LIN {X 0,Y 252.868,Z 364.586,A -85,B 0,C 180,E1 -18829.096,E2 -18829.096} C_VEL
LIN {X 0,Y 254.685,Z 356.199,A -85,B 0,C 180,E1 -18831.021,E2 -18831.021} C_VEL
LIN {X 0,Y 256.996,Z 345.688,A -85,B 0,C 180,E1 -18832.934,E2 -18832.934} C_VEL
LIN {X 0,Y 259.32,Z 333.859,A -85,B 0,C 180,E1 -18834.624,E2 -18834.624} C_VEL
LIN {X 0,Y 261.309,Z 321.945,A -85,B 0,C 180,E1 -18835.914,E2 -18835.914} C_VEL
LIN {X 0,Y 263.017,Z 309.547,A -85,B 0,C 180,E1 -18836.908,E2 -18836.908} C_VEL
LIN {X 0,Y 264.329,Z 296.774,A -85,B 0,C 180,E1 -18837.62,E2 -18837.62} C_VEL
LIN {X 0,Y 265.037,Z 283.246,A -85,B 0,C 180,E1 -18838.077,E2 -18838.077} C_VEL
LIN {X 0,Y 266.594,Z 234.638,A -85,B 0,C 180,E1 -18839.358,E2 -18839.358} C_VEL
LIN {X 0,Y 262.492,Z 206.676,A -85,B 0,C 180,E1 -18840.723,E2 -18840.723} C_VEL
LIN {X 0,Y 261.328,Z 202.665,A -85,B 0,C 180,E1 -18840.998,E2 -18840.998} C_VEL
LIN {X 0,Y 254.314,Z 186.379,A -85,B 0,C 180,E1 -18842.473,E2 -18842.473} C_VEL
LIN {X 0,Y 252.675,Z 182.594,A -85,B 0,C 180,E1 -18842.867,E2 -18842.867} C_VEL
LIN {X 0,Y 250.564,Z 173.371,A -85,B 0,C 180,E1 -18846.585,E2 -18846.585} C_VEL
LIN {X 0,Y 249.019,Z 167.461,A -85,B 0,C 180,E1 -18849.158,E2 -18849.158} C_VEL
LIN {X 0,Y 248.966,Z 167.471,A -85,B 0,C 180,E1 -18852.781,E2 -18852.781} C_VEL
LIN {X 0,Y 248.974,Z 167.471,A -85,B 0,C 180,E1 -18857.354,E2 -18857.354} C_VEL
LIN {X 0,Y 249.034,Z 167.462,A -85,B 0,C 180,E1 -18862.201,E2 -18862.201} C_VEL
LIN {X 0,Y 249.037,Z 167.461,A -85,B 0,C 180,E1 -18865.638,E2 -18865.638} C_VEL
LIN {X 0,Y 248.996,Z 167.466,A -85,B 0,C 180,E1 -18869.465,E2 -18869.465} C_VEL
LIN {X 0,Y 249.015,Z 167.464,A -85,B 0,C 180,E1 -18873.155,E2 -18873.155} C_VEL
LIN {X 0,Y 248.999,Z 167.459,A -85,B 0,C 180,E1 -18876.725,E2 -18876.725} C_VEL
LIN {X 0,Y 249.035,Z 167.464,A -85,B 0,C 180,E1 -18880.205,E2 -18880.205} C_VEL
LIN {X 0,Y 249.151,Z 167.437,A -85,B 0,C 180,E1 -18883.616,E2 -18883.616} C_VEL
LIN {X 0,Y 249.21,Z 167.436,A -85,B 0,C 180,E1 -18888.615,E2 -18888.615} C_VEL
LIN {X 0,Y 249.394,Z 167.413,A -85,B 0,C 180,E1 -18891.9,E2 -18891.9} C_VEL
LIN {X 0,Y 249.245,Z 167.435,A -85,B 0,C 180,E1 -18895.148,E2 -18895.148} C_VEL
LIN {X 0,Y 249.646,Z 167.378,A -85,B 0,C 180,E1 -18898.387,E2 -18898.387} C_VEL
LIN {X 0,Y 249.648,Z 167.388,A -85,B 0,C 180,E1 -18901.613,E2 -18901.613} C_VEL
LIN {X 0,Y 249.415,Z 167.411,A -85,B 0,C 180,E1 -18906.557,E2 -18906.557} C_VEL
LIN {X 0,Y 249.325,Z 167.427,A -85,B 0,C 180,E1 -18909.737,E2 -18909.737} C_VEL
LIN {X 0,Y 249.139,Z 167.448,A -85,B 0,C 180,E1 -18914.708,E2 -18914.708} C_VEL
LIN {X 0,Y 249.073,Z 167.452,A -85,B 0,C 180,E1 -18918.082,E2 -18918.082} C_VEL
LIN {X 0,Y 249.039,Z 167.461,A -85,B 0,C 180,E1 -18921.523,E2 -18921.523} C_VEL
LIN {X 0,Y 249.056,Z 167.452,A -85,B 0,C 180,E1 -18925.449,E2 -18925.449} C_VEL
LIN {X 0,Y 249.03,Z 167.466,A -85,B 0,C 180,E1 -18928.974,E2 -18928.974} C_VEL
LIN {X 0,Y 249.022,Z 167.458,A -85,B 0,C 180,E1 -18932.427,E2 -18932.427} C_VEL
LIN {X 0,Y 249.021,Z 167.465,A -85,B 0,C 180,E1 -18936.347,E2 -18936.347} C_VEL
LIN {X 0,Y 248.974,Z 167.47,A -85,B 0,C 180,E1 -18940.485,E2 -18940.485} C_VEL
LIN {X 0,Y 248.978,Z 167.466,A -85,B 0,C 180,E1 -18944.885,E2 -18944.885} C_VEL
LIN {X 0,Y 249.003,Z 167.467,A -85,B 0,C 180,E1 -18947.362,E2 -18947.362} C_VEL
LIN {X 0,Y 249.039,Z 167.461,A -85,B 0,C 180,E1 -18952.202,E2 -18952.202} C_VEL
LIN {X 0,Y 249.028,Z 167.546,A -85,B 0,C 180,E1 -18956.659,E2 -18956.659} C_VEL
LIN {X 0,Y 250.144,Z 170.47,A -85,B 0,C 180,E1 -18956.949,E2 -18956.949} C_VEL
LIN {X 0,Y 251.527,Z 172.737,A -85,B 0,C 180,E1 -18957.231,E2 -18957.231} C_VEL
LIN {X 0,Y 257.093,Z 183.362,A -85,B 0,C 180,E1 -18958.378,E2 -18958.378} C_VEL
LIN {X 0,Y 264.699,Z 200.479,A -85,B 0,C 180,E1 -18959.926,E2 -18959.926} C_VEL
LIN {X 0,Y 267.489,Z 207.786,A -85,B 0,C 180,E1 -18960.497,E2 -18960.497} C_VEL
LIN {X 0,Y 265.356,Z 271.347,A -85,B 0,C 180,E1 -18962.177,E2 -18962.177} C_VEL
LIN {X 0,Y 264.517,Z 284.387,A -85,B 0,C 180,E1 -18962.724,E2 -18962.724} C_VEL
LIN {X 0,Y 263.3,Z 296.87,A -85,B 0,C 180,E1 -18963.551,E2 -18963.551} C_VEL
LIN {X 0,Y 261.894,Z 308.06,A -85,B 0,C 180,E1 -18964.574,E2 -18964.574} C_VEL
LIN {X 0,Y 260.057,Z 319.137,A -85,B 0,C 180,E1 -18965.875,E2 -18965.875} C_VEL
LIN {X 0,Y 258.172,Z 329.268,A -85,B 0,C 180,E1 -18967.388,E2 -18967.388} C_VEL
LIN {X 0,Y 256.493,Z 338.564,A -85,B 0,C 180,E1 -18969.134,E2 -18969.134} C_VEL
LIN {X 0,Y 254.459,Z 347.043,A -85,B 0,C 180,E1 -18971.064,E2 -18971.064} C_VEL
LIN {X 0,Y 252.372,Z 355.282,A -85,B 0,C 180,E1 -18973.416,E2 -18973.416} C_VEL
LIN {X 0,Y 250.964,Z 360.914,A -85,B 0,C 180,E1 -18975.403,E2 -18975.403} C_VEL
LIN {X 0,Y 249.579,Z 366.401,A -85,B 0,C 180,E1 -18977.809,E2 -18977.809} C_VEL
LIN {X 0,Y 248.492,Z 370.708,A -85,B 0,C 180,E1 -18980.231,E2 -18980.231} C_VEL
LIN {X 0,Y 247.724,Z 374.525,A -85,B 0,C 180,E1 -18983.2,E2 -18983.2} C_VEL
LIN {X 0,Y 247.414,Z 376.22,A -85,B 0,C 180,E1 -18985.112,E2 -18985.112} C_VEL
LIN {X 0,Y 247.22,Z 377.209,A -85,B 0,C 180,E1 -18986.742,E2 -18986.742} C_VEL
LIN {X 0,Y 247.041,Z 378.047,A -85,B 0,C 180,E1 -18990.001,E2 -18990.001} C_VEL
LIN {X 0,Y 247.079,Z 377.854,A -85,B 0,C 180,E1 -18991.631,E2 -18991.631} C_VEL
LIN {X 0,Y 247.218,Z 377.268,A -85,B 0,C 180,E1 -18993.26,E2 -18993.26} C_VEL
LIN {X 0,Y 247.408,Z 376.303,A -85,B 0,C 180,E1 -18994.889,E2 -18994.889} C_VEL
LIN {X 0,Y 247.716,Z 374.678,A -85,B 0,C 180,E1 -18996.784,E2 -18996.784} C_VEL
LIN {X 0,Y 248.467,Z 370.899,A -85,B 0,C 180,E1 -18999.772,E2 -18999.772} C_VEL
LIN {X 0,Y 249.523,Z 366.652,A -85,B 0,C 180,E1 -19002.196,E2 -19002.196} C_VEL
LIN {X 0,Y 251.213,Z 360.217,A -85,B 0,C 180,E1 -19004.998,E2 -19004.998} C_VEL
LIN {X 0,Y 252.923,Z 353.147,A -85,B 0,C 180,E1 -19007.381,E2 -19007.381} C_VEL
LIN {X 0,Y 255.176,Z 344.328,A -85,B 0,C 180,E1 -19009.718,E2 -19009.718} C_VEL
LIN {X 0,Y 257.073,Z 335.367,A -85,B 0,C 180,E1 -19011.641,E2 -19011.641} C_VEL
LIN {X 0,Y 259.036,Z 325.258,A -85,B 0,C 180,E1 -19013.379,E2 -19013.379} C_VEL
LIN {X 0,Y 261.004,Z 314.1,A -85,B 0,C 180,E1 -19014.881,E2 -19014.881} C_VEL
LIN {X 0,Y 262.591,Z 303.55,A -85,B 0,C 180,E1 -19015.993,E2 -19015.993} C_VEL
LIN {X 0,Y 264.079,Z 290.832,A -85,B 0,C 180,E1 -19017.007,E2 -19017.007} C_VEL
LIN {X 0,Y 265.098,Z 278.105,A -85,B 0,C 180,E1 -19017.696,E2 -19017.696} C_VEL
LIN {X 0,Y 265.964,Z 260.051,A -85,B 0,C 180,E1 -19018.24,E2 -19018.24} C_VEL
LIN {X 0,Y 267.533,Z 207.816,A -85,B 0,C 180,E1 -19019.63,E2 -19019.63} C_VEL
LIN {X 0,Y 261.17,Z 192.177,A -85,B 0,C 180,E1 -19020.926,E2 -19020.926} C_VEL
LIN {X 0,Y 254.413,Z 178.027,A -85,B 0,C 180,E1 -19022.313,E2 -19022.313} C_VEL
LIN {X 0,Y 250.64,Z 171.151,A -85,B 0,C 180,E1 -19023.096,E2 -19023.096} C_VEL
LIN {X 0,Y 249.295,Z 168.69,A -85,B 0,C 180,E1 -19023.383,E2 -19023.383} C_VEL
LIN {X 0,Y 249.029,Z 167.477,A -85,B 0,C 180,E1 -19023.515,E2 -19023.515} C_VEL
LIN {X 0,Y 249.04,Z 167.465,A -85,B 0,C 180,E1 -19027.798,E2 -19027.798} C_VEL
LIN {X 0,Y 248.978,Z 167.471,A -85,B 0,C 180,E1 -19032.646,E2 -19032.646} C_VEL
LIN {X 0,Y 248.98,Z 167.471,A -85,B 0,C 180,E1 -19037.355,E2 -19037.355} C_VEL
LIN {X 0,Y 249.041,Z 167.461,A -85,B 0,C 180,E1 -19042.201,E2 -19042.201} C_VEL
LIN {X 0,Y 249.044,Z 167.456,A -85,B 0,C 180,E1 -19045.639,E2 -19045.639} C_VEL
LIN {X 0,Y 249.003,Z 167.462,A -85,B 0,C 180,E1 -19049.466,E2 -19049.466} C_VEL
LIN {X 0,Y 249.036,Z 167.465,A -85,B 0,C 180,E1 -19053.158,E2 -19053.158} C_VEL
LIN {X 0,Y 249.056,Z 167.45,A -85,B 0,C 180,E1 -19056.73,E2 -19056.73} C_VEL
LIN {X 0,Y 249.076,Z 167.457,A -85,B 0,C 180,E1 -19060.208,E2 -19060.208} C_VEL
LIN {X 0,Y 249.158,Z 167.441,A -85,B 0,C 180,E1 -19063.616,E2 -19063.616} C_VEL
LIN {X 0,Y 249.229,Z 167.441,A -85,B 0,C 180,E1 -19068.615,E2 -19068.615} C_VEL
LIN {X 0,Y 249.417,Z 167.405,A -85,B 0,C 180,E1 -19071.901,E2 -19071.901} C_VEL
LIN {X 0,Y 249.258,Z 167.431,A -85,B 0,C 180,E1 -19075.148,E2 -19075.148} C_VEL
LIN {X 0,Y 249.655,Z 167.384,A -85,B 0,C 180,E1 -19078.387,E2 -19078.387} C_VEL
LIN {X 0,Y 249.653,Z 167.37,A -85,B 0,C 180,E1 -19081.613,E2 -19081.613} C_VEL
LIN {X 0,Y 249.252,Z 167.435,A -85,B 0,C 180,E1 -19084.802,E2 -19084.802} C_VEL
LIN {X 0,Y 248.58,Z 167.529,A -85,B 0,C 180,E1 -19086.153,E2 -19086.153} C_VEL
LIN {X 0,Y 245.744,Z 167.883,A -85,B 0,C 180,E1 -19088.356,E2 -19088.356} C_VEL
LIN {X 0,Y 243.315,Z 168.178,A -85,B 0,C 180,E1 -19090.15,E2 -19090.15} C_VEL
LIN {X 0,Y 242.234,Z 168.307,A -85,B 0,C 180,E1 -19091.541,E2 -19091.541} C_VEL
LIN {X 0,Y 242.125,Z 168.319,A -85,B 0,C 180,E1 -19092.013,E2 -19092.013} C_VEL
LIN {X 0,Y 242.092,Z 168.312,A -85,B 0,C 180,E1 -19096.876,E2 -19096.876} C_VEL
LIN {X 0,Y 241.972,Z 168.336,A -85,B 0,C 180,E1 -19102.184,E2 -19102.184} C_VEL
LIN {X 0,Y 241.987,Z 168.342,A -85,B 0,C 180,E1 -19105.826,E2 -19105.826} C_VEL
LIN {X 0,Y 241.968,Z 168.337,A -85,B 0,C 180,E1 -19109.589,E2 -19109.589} C_VEL
LIN {X 0,Y 241.98,Z 168.335,A -85,B 0,C 180,E1 -19113.493,E2 -19113.493} C_VEL
LIN {X 0,Y 241.978,Z 168.336,A -85,B 0,C 180,E1 -19117.584,E2 -19117.584} C_VEL
LIN {X 0,Y 241.908,Z 168.347,A -85,B 0,C 180,E1 -19121.929,E2 -19121.929} C_VEL
LIN {X 0,Y 241.901,Z 168.351,A -85,B 0,C 180,E1 -19126.58,E2 -19126.58} C_VEL
LIN {X 0,Y 241.977,Z 168.45,A -85,B 0,C 180,E1 -19129.989,E2 -19129.989} C_VEL
LIN {X 0,Y 244.385,Z 177.67,A -85,B 0,C 180,E1 -19134.066,E2 -19134.066} C_VEL
LIN {X 0,Y 245.43,Z 182.458,A -85,B 0,C 180,E1 -19136.022,E2 -19136.022} C_VEL
LIN {X 0,Y 253.06,Z 199.303,A -85,B 0,C 180,E1 -19137.723,E2 -19137.723} C_VEL
LIN {X 0,Y 256.555,Z 208.314,A -85,B 0,C 180,E1 -19138.499,E2 -19138.499} C_VEL
LIN {X 0,Y 260.098,Z 232.626,A -85,B 0,C 180,E1 -19139.735,E2 -19139.735} C_VEL
LIN {X 0,Y 260.446,Z 237.003,A -85,B 0,C 180,E1 -19139.915,E2 -19139.915} C_VEL
LIN {X 0,Y 258.519,Z 291.741,A -85,B 0,C 180,E1 -19141.425,E2 -19141.425} C_VEL
LIN {X 0,Y 257.264,Z 305.637,A -85,B 0,C 180,E1 -19142.106,E2 -19142.106} C_VEL
LIN {X 0,Y 255.612,Z 318.073,A -85,B 0,C 180,E1 -19143.021,E2 -19143.021} C_VEL
LIN {X 0,Y 253.774,Z 329.173,A -85,B 0,C 180,E1 -19144.139,E2 -19144.139} C_VEL
LIN {X 0,Y 251.513,Z 340.745,A -85,B 0,C 180,E1 -19145.659,E2 -19145.659} C_VEL
LIN {X 0,Y 249.22,Z 351.171,A -85,B 0,C 180,E1 -19147.404,E2 -19147.404} C_VEL
LIN {X 0,Y 247.242,Z 359.7,A -85,B 0,C 180,E1 -19149.186,E2 -19149.186} C_VEL
LIN {X 0,Y 245.437,Z 367.793,A -85,B 0,C 180,E1 -19151.272,E2 -19151.272} C_VEL
LIN {X 0,Y 243.537,Z 375.272,A -85,B 0,C 180,E1 -19153.658,E2 -19153.658} C_VEL
LIN {X 0,Y 241.694,Z 382.371,A -85,B 0,C 180,E1 -19156.548,E2 -19156.548} C_VEL
LIN {X 0,Y 240.787,Z 387.105,A -85,B 0,C 180,E1 -19159.063,E2 -19159.063} C_VEL
LIN {X 0,Y 240.158,Z 390.724,A -85,B 0,C 180,E1 -19161.585,E2 -19161.585} C_VEL
LIN {X 0,Y 239.899,Z 392.592,A -85,B 0,C 180,E1 -19163.27,E2 -19163.27} C_VEL
LIN {X 0,Y 239.798,Z 394.153,A -85,B 0,C 180,E1 -19165.188,E2 -19165.188} C_VEL
LIN {X 0,Y 239.883,Z 395.614,A -85,B 0,C 180,E1 -19168.32,E2 -19168.32} C_VEL
LIN {X 0,Y 239.956,Z 395.83,A -85,B 0,C 180,E1 -19169.999,E2 -19169.999} C_VEL
LIN {X 0,Y 239.883,Z 395.604,A -85,B 0,C 180,E1 -19171.678,E2 -19171.678} C_VEL
LIN {X 0,Y 239.78,Z 394.165,A -85,B 0,C 180,E1 -19174.76,E2 -19174.76} C_VEL
LIN {X 0,Y 239.905,Z 392.559,A -85,B 0,C 180,E1 -19176.728,E2 -19176.728} C_VEL
LIN {X 0,Y 240.359,Z 389.6,A -85,B 0,C 180,E1 -19179.253,E2 -19179.253} C_VEL
LIN {X 0,Y 241.052,Z 385.599,A -85,B 0,C 180,E1 -19181.775,E2 -19181.775} C_VEL
LIN {X 0,Y 242.451,Z 379.459,A -85,B 0,C 180,E1 -19184.692,E2 -19184.692} C_VEL
LIN {X 0,Y 244.066,Z 372.759,A -85,B 0,C 180,E1 -19187.166,E2 -19187.166} C_VEL
LIN {X 0,Y 245.951,Z 365.05,A -85,B 0,C 180,E1 -19189.444,E2 -19189.444} C_VEL
LIN {X 0,Y 248.049,Z 355.936,A -85,B 0,C 180,E1 -19191.611,E2 -19191.611} C_VEL
LIN {X 0,Y 250.431,Z 345.424,A -85,B 0,C 180,E1 -19193.571,E2 -19193.571} C_VEL
LIN {X 0,Y 252.885,Z 333.595,A -85,B 0,C 180,E1 -19195.294,E2 -19195.294} C_VEL
LIN {X 0,Y 254.951,Z 321.68,A -85,B 0,C 180,E1 -19196.611,E2 -19196.611} C_VEL
LIN {X 0,Y 256.725,Z 309.281,A -85,B 0,C 180,E1 -19197.623,E2 -19197.623} C_VEL
LIN {X 0,Y 258.064,Z 296.503,A -85,B 0,C 180,E1 -19198.35,E2 -19198.35} C_VEL
LIN {X 0,Y 258.784,Z 282.965,A -85,B 0,C 180,E1 -19198.818,E2 -19198.818} C_VEL
LIN {X 0,Y 260.307,Z 234.676,A -85,B 0,C 180,E1 -19200.13,E2 -19200.13} C_VEL
LIN {X 0,Y 256.425,Z 208.257,A -85,B 0,C 180,E1 -19201.472,E2 -19201.472} C_VEL
LIN {X 0,Y 254.062,Z 201.684,A -85,B 0,C 180,E1 -19202.009,E2 -19202.009} C_VEL
LIN {X 0,Y 246.909,Z 185.778,A -85,B 0,C 180,E1 -19203.582,E2 -19203.582} C_VEL
LIN {X 0,Y 245.392,Z 182.189,A -85,B 0,C 180,E1 -19204.005,E2 -19204.005} C_VEL
LIN {X 0,Y 243.08,Z 172.44,A -85,B 0,C 180,E1 -19208.142,E2 -19208.142} C_VEL
LIN {X 0,Y 241.946,Z 168.341,A -85,B 0,C 180,E1 -19210.074,E2 -19210.074} C_VEL
LIN {X 0,Y 241.892,Z 168.354,A -85,B 0,C 180,E1 -19214.209,E2 -19214.209} C_VEL
LIN {X 0,Y 241.903,Z 168.353,A -85,B 0,C 180,E1 -19218.07,E2 -19218.07} C_VEL
LIN {X 0,Y 241.977,Z 168.34,A -85,B 0,C 180,E1 -19222.416,E2 -19222.416} C_VEL
LIN {X 0,Y 241.973,Z 168.337,A -85,B 0,C 180,E1 -19226.506,E2 -19226.506} C_VEL
LIN {X 0,Y 241.971,Z 168.337,A -85,B 0,C 180,E1 -19230.612,E2 -19230.612} C_VEL
LIN {X 0,Y 241.99,Z 168.339,A -85,B 0,C 180,E1 -19234.196,E2 -19234.196} C_VEL
LIN {X 0,Y 241.978,Z 168.335,A -85,B 0,C 180,E1 -19238.338,E2 -19238.338} C_VEL
LIN {X 0,Y 242.099,Z 168.314,A -85,B 0,C 180,E1 -19243.324,E2 -19243.324} C_VEL
LIN {X 0,Y 242.144,Z 168.318,A -85,B 0,C 180,E1 -19248.278,E2 -19248.278} C_VEL
LIN {X 0,Y 242.35,Z 168.289,A -85,B 0,C 180,E1 -19251.663,E2 -19251.663} C_VEL
LIN {X 0,Y 242.382,Z 168.291,A -85,B 0,C 180,E1 -19253.34,E2 -19253.34} C_VEL
LIN {X 0,Y 242.606,Z 168.254,A -85,B 0,C 180,E1 -19258.34,E2 -19258.34} C_VEL
LIN {X 0,Y 242.608,Z 168.266,A -85,B 0,C 180,E1 -19261.66,E2 -19261.66} C_VEL
LIN {X 0,Y 242.392,Z 168.286,A -85,B 0,C 180,E1 -19266.66,E2 -19266.66} C_VEL
LIN {X 0,Y 242.253,Z 168.306,A -85,B 0,C 180,E1 -19270.024,E2 -19270.024} C_VEL
LIN {X 0,Y 242.097,Z 168.326,A -85,B 0,C 180,E1 -19275.145,E2 -19275.145} C_VEL
LIN {X 0,Y 242.012,Z 168.331,A -85,B 0,C 180,E1 -19278.629,E2 -19278.629} C_VEL
LIN {X 0,Y 241.978,Z 168.342,A -85,B 0,C 180,E1 -19282.183,E2 -19282.183} C_VEL
LIN {X 0,Y 241.987,Z 168.33,A -85,B 0,C 180,E1 -19285.826,E2 -19285.826} C_VEL
LIN {X 0,Y 241.963,Z 168.344,A -85,B 0,C 180,E1 -19289.589,E2 -19289.589} C_VEL
LIN {X 0,Y 241.974,Z 168.344,A -85,B 0,C 180,E1 -19293.494,E2 -19293.494} C_VEL
LIN {X 0,Y 241.978,Z 168.341,A -85,B 0,C 180,E1 -19297.584,E2 -19297.584} C_VEL
LIN {X 0,Y 241.908,Z 168.35,A -85,B 0,C 180,E1 -19301.929,E2 -19301.929} C_VEL
LIN {X 0,Y 241.919,Z 168.35,A -85,B 0,C 180,E1 -19306.575,E2 -19306.575} C_VEL
LIN {X 0,Y 241.991,Z 168.337,A -85,B 0,C 180,E1 -19311.642,E2 -19311.642} C_VEL
LIN {X 0,Y 242.041,Z 168.531,A -85,B 0,C 180,E1 -19315.609,E2 -19315.609} C_VEL
LIN {X 0,Y 243.04,Z 171.272,A -85,B 0,C 180,E1 -19315.868,E2 -19315.868} C_VEL
LIN {X 0,Y 244.462,Z 173.486,A -85,B 0,C 180,E1 -19316.173,E2 -19316.173} C_VEL
LIN {X 0,Y 249.703,Z 182.957,A -85,B 0,C 180,E1 -19317.302,E2 -19317.302} C_VEL
LIN {X 0,Y 256.513,Z 197.662,A -85,B 0,C 180,E1 -19318.758,E2 -19318.758} C_VEL
LIN {X 0,Y 261.307,Z 209.496,A -85,B 0,C 180,E1 -19319.771,E2 -19319.771} C_VEL
LIN {X 0,Y 259.135,Z 271.055,A -85,B 0,C 180,E1 -19321.428,E2 -19321.428} C_VEL
LIN {X 0,Y 258.314,Z 283.988,A -85,B 0,C 180,E1 -19321.971,E2 -19321.971} C_VEL
LIN {X 0,Y 257.098,Z 295.986,A -85,B 0,C 180,E1 -19322.751,E2 -19322.751} C_VEL
LIN {X 0,Y 255.523,Z 308.324,A -85,B 0,C 180,E1 -19323.893,E2 -19323.893} C_VEL
LIN {X 0,Y 253.592,Z 319.401,A -85,B 0,C 180,E1 -19325.219,E2 -19325.219} C_VEL
LIN {X 0,Y 251.628,Z 329.532,A -85,B 0,C 180,E1 -19326.766,E2 -19326.766} C_VEL
LIN {X 0,Y 249.869,Z 338.826,A -85,B 0,C 180,E1 -19328.554,E2 -19328.554} C_VEL
LIN {X 0,Y 247.752,Z 347.304,A -85,B 0,C 180,E1 -19330.531,E2 -19330.531} C_VEL
LIN {X 0,Y 245.588,Z 355.543,A -85,B 0,C 180,E1 -19332.944,E2 -19332.944} C_VEL
LIN {X 0,Y 244.098,Z 361.175,A -85,B 0,C 180,E1 -19334.983,E2 -19334.983} C_VEL
LIN {X 0,Y 242.646,Z 366.662,A -85,B 0,C 180,E1 -19337.455,E2 -19337.455} C_VEL
LIN {X 0,Y 241.503,Z 370.968,A -85,B 0,C 180,E1 -19339.945,E2 -19339.945} C_VEL
LIN {X 0,Y 240.976,Z 373.243,A -85,B 0,C 180,E1 -19341.616,E2 -19341.616} C_VEL
LIN {X 0,Y 240.601,Z 375.091,A -85,B 0,C 180,E1 -19343.291,E2 -19343.291} C_VEL
LIN {X 0,Y 240.334,Z 376.48,A -85,B 0,C 180,E1 -19344.968,E2 -19344.968} C_VEL
LIN {X 0,Y 240.142,Z 377.468,A -85,B 0,C 180,E1 -19346.645,E2 -19346.645} C_VEL
LIN {X 0,Y 239.971,Z 378.305,A -85,B 0,C 180,E1 -19350.001,E2 -19350.001} C_VEL
LIN {X 0,Y 240.012,Z 378.112,A -85,B 0,C 180,E1 -19351.679,E2 -19351.679} C_VEL
LIN {X 0,Y 240.139,Z 377.527,A -85,B 0,C 180,E1 -19353.356,E2 -19353.356} C_VEL
LIN {X 0,Y 240.329,Z 376.562,A -85,B 0,C 180,E1 -19355.034,E2 -19355.034} C_VEL
LIN {X 0,Y 240.602,Z 375.209,A -85,B 0,C 180,E1 -19356.711,E2 -19356.711} C_VEL
LIN {X 0,Y 241.197,Z 372.35,A -85,B 0,C 180,E1 -19359.223,E2 -19359.223} C_VEL
LIN {X 0,Y 242.16,Z 368.467,A -85,B 0,C 180,E1 -19361.722,E2 -19361.722} C_VEL
LIN {X 0,Y 243.536,Z 363.454,A -85,B 0,C 180,E1 -19364.2,E2 -19364.2} C_VEL
LIN {X 0,Y 245.157,Z 357.141,A -85,B 0,C 180,E1 -19366.66,E2 -19366.66} C_VEL
LIN {X 0,Y 247.326,Z 349.232,A -85,B 0,C 180,E1 -19369.074,E2 -19369.074} C_VEL
LIN {X 0,Y 249.737,Z 339.396,A -85,B 0,C 180,E1 -19371.46,E2 -19371.46} C_VEL
LIN {X 0,Y 251.803,Z 329.072,A -85,B 0,C 180,E1 -19373.437,E2 -19373.437} C_VEL
LIN {X 0,Y 254.091,Z 317.414,A -85,B 0,C 180,E1 -19375.168,E2 -19375.168} C_VEL
LIN {X 0,Y 256.028,Z 305.781,A -85,B 0,C 180,E1 -19376.492,E2 -19376.492} C_VEL
LIN {X 0,Y 257.504,Z 293.679,A -85,B 0,C 180,E1 -19377.534,E2 -19377.534} C_VEL
LIN {X 0,Y 258.64,Z 281.366,A -85,B 0,C 180,E1 -19378.284,E2 -19378.284} C_VEL
LIN {X 0,Y 259.432,Z 269.158,A -85,B 0,C 180,E1 -19378.741,E2 -19378.741} C_VEL
LIN {X 0,Y 261.376,Z 209.619,A -85,B 0,C 180,E1 -19380.352,E2 -19380.352} C_VEL
LIN {X 0,Y 254.384,Z 192.715,A -85,B 0,C 180,E1 -19381.837,E2 -19381.837} C_VEL
LIN {X 0,Y 247.191,Z 178.132,A -85,B 0,C 180,E1 -19383.385,E2 -19383.385} C_VEL
LIN {X 0,Y 243.415,Z 171.757,A -85,B 0,C 180,E1 -19384.201,E2 -19384.201} C_VEL
LIN {X 0,Y 242.12,Z 168.986,A -85,B 0,C 180,E1 -19384.509,E2 -19384.509} C_VEL
LIN {X 0,Y 242.017,Z 168.336,A -85,B 0,C 180,E1 -19384.643,E2 -19384.643} C_VEL
LIN {X 0,Y 241.986,Z 168.342,A -85,B 0,C 180,E1 -19388.356,E2 -19388.356} C_VEL
LIN {X 0,Y 241.9,Z 168.354,A -85,B 0,C 180,E1 -19393.42,E2 -19393.42} C_VEL
LIN {X 0,Y 241.909,Z 168.35,A -85,B 0,C 180,E1 -19398.071,E2 -19398.071} C_VEL
LIN {X 0,Y 241.984,Z 168.341,A -85,B 0,C 180,E1 -19402.417,E2 -19402.417} C_VEL
LIN {X 0,Y 241.98,Z 168.338,A -85,B 0,C 180,E1 -19406.507,E2 -19406.507} C_VEL
LIN {X 0,Y 241.978,Z 168.332,A -85,B 0,C 180,E1 -19410.613,E2 -19410.613} C_VEL
LIN {X 0,Y 242.033,Z 168.336,A -85,B 0,C 180,E1 -19414.179,E2 -19414.179} C_VEL
LIN {X 0,Y 242.023,Z 168.324,A -85,B 0,C 180,E1 -19418.316,E2 -19418.316} C_VEL
LIN {X 0,Y 242.106,Z 168.319,A -85,B 0,C 180,E1 -19423.324,E2 -19423.324} C_VEL
LIN {X 0,Y 242.161,Z 168.32,A -85,B 0,C 180,E1 -19428.278,E2 -19428.278} C_VEL
LIN {X 0,Y 242.371,Z 168.284,A -85,B 0,C 180,E1 -19431.664,E2 -19431.664} C_VEL
LIN {X 0,Y 242.395,Z 168.273,A -85,B 0,C 180,E1 -19433.34,E2 -19433.34} C_VEL
LIN {X 0,Y 242.615,Z 168.261,A -85,B 0,C 180,E1 -19438.34,E2 -19438.34} C_VEL
LIN {X 0,Y 242.613,Z 168.246,A -85,B 0,C 180,E1 -19441.66,E2 -19441.66} C_VEL
LIN {X 0,Y 242.389,Z 168.288,A -85,B 0,C 180,E1 -19446.66,E2 -19446.66} C_VEL
LIN {X 0,Y 242.259,Z 168.293,A -85,B 0,C 180,E1 -19450.024,E2 -19450.024} C_VEL
LIN {X 0,Y 242.125,Z 168.319,A -85,B 0,C 180,E1 -19452.013,E2 -19452.013} C_VEL
LIN {X 0,Y 241.405,Z 168.414,A -85,B 0,C 180,E1 -19453.401,E2 -19453.401} C_VEL
LIN {X 0,Y 238.542,Z 168.77,A -85,B 0,C 180,E1 -19455.667,E2 -19455.667} C_VEL
LIN {X 0,Y 236.119,Z 169.073,A -85,B 0,C 180,E1 -19457.513,E2 -19457.513} C_VEL
LIN {X 0,Y 235.046,Z 169.204,A -85,B 0,C 180,E1 -19458.944,E2 -19458.944} C_VEL
LIN {X 0,Y 234.939,Z 169.216,A -85,B 0,C 180,E1 -19459.43,E2 -19459.43} C_VEL
LIN {X 0,Y 234.908,Z 169.212,A -85,B 0,C 180,E1 -19462.888,E2 -19462.888} C_VEL
LIN {X 0,Y 234.925,Z 169.221,A -85,B 0,C 180,E1 -19466.663,E2 -19466.663} C_VEL
LIN {X 0,Y 234.899,Z 169.222,A -85,B 0,C 180,E1 -19470.573,E2 -19470.573} C_VEL
LIN {X 0,Y 234.925,Z 169.215,A -85,B 0,C 180,E1 -19474.639,E2 -19474.639} C_VEL
LIN {X 0,Y 234.913,Z 169.219,A -85,B 0,C 180,E1 -19478.935,E2 -19478.935} C_VEL
LIN {X 0,Y 234.854,Z 169.23,A -85,B 0,C 180,E1 -19483.494,E2 -19483.494} C_VEL
LIN {X 0,Y 234.854,Z 169.229,A -85,B 0,C 180,E1 -19486.506,E2 -19486.506} C_VEL
LIN {X 0,Y 234.902,Z 169.352,A -85,B 0,C 180,E1 -19489.054,E2 -19489.054} C_VEL
LIN {X 0,Y 236.86,Z 176.598,A -85,B 0,C 180,E1 -19492.435,E2 -19492.435} C_VEL
LIN {X 0,Y 238.232,Z 182.249,A -85,B 0,C 180,E1 -19494.85,E2 -19494.85} C_VEL
LIN {X 0,Y 246.011,Z 199.023,A -85,B 0,C 180,E1 -19496.68,E2 -19496.68} C_VEL
LIN {X 0,Y 250.572,Z 210.141,A -85,B 0,C 180,E1 -19497.726,E2 -19497.726} C_VEL
LIN {X 0,Y 253.989,Z 233.847,A -85,B 0,C 180,E1 -19498.974,E2 -19498.974} C_VEL
LIN {X 0,Y 254.258,Z 238.85,A -85,B 0,C 180,E1 -19499.171,E2 -19499.171} C_VEL
LIN {X 0,Y 252.301,Z 291.495,A -85,B 0,C 180,E1 -19500.653,E2 -19500.653} C_VEL
LIN {X 0,Y 251.015,Z 305.387,A -85,B 0,C 180,E1 -19501.349,E2 -19501.349} C_VEL
LIN {X 0,Y 249.297,Z 317.82,A -85,B 0,C 180,E1 -19502.279,E2 -19502.279} C_VEL
LIN {X 0,Y 247.387,Z 328.918,A -85,B 0,C 180,E1 -19503.42,E2 -19503.42} C_VEL
LIN {X 0,Y 245.049,Z 340.489,A -85,B 0,C 180,E1 -19504.973,E2 -19504.973} C_VEL
LIN {X 0,Y 242.668,Z 350.914,A -85,B 0,C 180,E1 -19506.758,E2 -19506.758} C_VEL
LIN {X 0,Y 240.571,Z 359.442,A -85,B 0,C 180,E1 -19508.581,E2 -19508.581} C_VEL
LIN {X 0,Y 238.792,Z 366.931,A -85,B 0,C 180,E1 -19510.546,E2 -19510.546} C_VEL
LIN {X 0,Y 236.67,Z 375.012,A -85,B 0,C 180,E1 -19513.17,E2 -19513.17} C_VEL
LIN {X 0,Y 234.769,Z 382.112,A -85,B 0,C 180,E1 -19516.143,E2 -19516.143} C_VEL
LIN {X 0,Y 233.779,Z 386.846,A -85,B 0,C 180,E1 -19518.731,E2 -19518.731} C_VEL
LIN {X 0,Y 233.109,Z 390.465,A -85,B 0,C 180,E1 -19521.329,E2 -19521.329} C_VEL
LIN {X 0,Y 232.821,Z 392.332,A -85,B 0,C 180,E1 -19523.064,E2 -19523.064} C_VEL
LIN {X 0,Y 232.702,Z 394.075,A -85,B 0,C 180,E1 -19525.315,E2 -19525.315} C_VEL
LIN {X 0,Y 232.792,Z 395.355,A -85,B 0,C 180,E1 -19528.269,E2 -19528.269} C_VEL
LIN {X 0,Y 232.886,Z 395.572,A -85,B 0,C 180,E1 -19529.999,E2 -19529.999} C_VEL
LIN {X 0,Y 232.792,Z 395.345,A -85,B 0,C 180,E1 -19531.729,E2 -19531.729} C_VEL
LIN {X 0,Y 232.729,Z 393.713,A -85,B 0,C 180,E1 -19535.197,E2 -19535.197} C_VEL
LIN {X 0,Y 232.827,Z 392.298,A -85,B 0,C 180,E1 -19536.934,E2 -19536.934} C_VEL
LIN {X 0,Y 233.307,Z 389.339,A -85,B 0,C 180,E1 -19539.536,E2 -19539.536} C_VEL
LIN {X 0,Y 234.05,Z 385.337,A -85,B 0,C 180,E1 -19542.133,E2 -19542.133} C_VEL
LIN {X 0,Y 235.54,Z 379.196,A -85,B 0,C 180,E1 -19545.133,E2 -19545.133} C_VEL
LIN {X 0,Y 237.274,Z 372.497,A -85,B 0,C 180,E1 -19547.673,E2 -19547.673} C_VEL
LIN {X 0,Y 239.518,Z 363.714,A -85,B 0,C 180,E1 -19550.306,E2 -19550.306} C_VEL
LIN {X 0,Y 241.435,Z 355.673,A -85,B 0,C 180,E1 -19552.235,E2 -19552.235} C_VEL
LIN {X 0,Y 243.9,Z 345.159,A -85,B 0,C 180,E1 -19554.242,E2 -19554.242} C_VEL
LIN {X 0,Y 246.478,Z 333.332,A -85,B 0,C 180,E1 -19556,E2 -19556} C_VEL
LIN {X 0,Y 248.639,Z 321.415,A -85,B 0,C 180,E1 -19557.342,E2 -19557.342} C_VEL
LIN {X 0,Y 250.469,Z 309.014,A -85,B 0,C 180,E1 -19558.375,E2 -19558.375} C_VEL
LIN {X 0,Y 251.815,Z 296.514,A -85,B 0,C 180,E1 -19559.104,E2 -19559.104} C_VEL
LIN {X 0,Y 252.599,Z 281.83,A -85,B 0,C 180,E1 -19559.62,E2 -19559.62} C_VEL
LIN {X 0,Y 254.17,Z 235.706,A -85,B 0,C 180,E1 -19560.894,E2 -19560.894} C_VEL
LIN {X 0,Y 250.48,Z 210.128,A -85,B 0,C 180,E1 -19562.237,E2 -19562.237} C_VEL
LIN {X 0,Y 244.956,Z 196.69,A -85,B 0,C 180,E1 -19563.507,E2 -19563.507} C_VEL
LIN {X 0,Y 238.823,Z 183.808,A -85,B 0,C 180,E1 -19564.936,E2 -19564.936} C_VEL
LIN {X 0,Y 238.136,Z 182.052,A -85,B 0,C 180,E1 -19565.119,E2 -19565.119} C_VEL
LIN {X 0,Y 236.193,Z 174.038,A -85,B 0,C 180,E1 -19568.67,E2 -19568.67} C_VEL
LIN {X 0,Y 234.872,Z 169.225,A -85,B 0,C 180,E1 -19570.95,E2 -19570.95} C_VEL
LIN {X 0,Y 234.858,Z 169.23,A -85,B 0,C 180,E1 -19574.095,E2 -19574.095} C_VEL
LIN {X 0,Y 234.849,Z 169.23,A -85,B 0,C 180,E1 -19578.825,E2 -19578.825} C_VEL
LIN {X 0,Y 234.913,Z 169.225,A -85,B 0,C 180,E1 -19581.078,E2 -19581.078} C_VEL
LIN {X 0,Y 234.919,Z 169.22,A -85,B 0,C 180,E1 -19585.36,E2 -19585.36} C_VEL
LIN {X 0,Y 234.893,Z 169.223,A -85,B 0,C 180,E1 -19589.427,E2 -19589.427} C_VEL
LIN {X 0,Y 234.934,Z 169.217,A -85,B 0,C 180,E1 -19593.82,E2 -19593.82} C_VEL
LIN {X 0,Y 234.929,Z 169.219,A -85,B 0,C 180,E1 -19598.962,E2 -19598.962} C_VEL
LIN {X 0,Y 235.043,Z 169.193,A -85,B 0,C 180,E1 -19603.097,E2 -19603.097} C_VEL
LIN {X 0,Y 235.076,Z 169.202,A -85,B 0,C 180,E1 -19607.92,E2 -19607.92} C_VEL
LIN {X 0,Y 235.288,Z 169.168,A -85,B 0,C 180,E1 -19611.411,E2 -19611.411} C_VEL
LIN {X 0,Y 235.333,Z 169.169,A -85,B 0,C 180,E1 -19613.139,E2 -19613.139} C_VEL
LIN {X 0,Y 235.565,Z 169.13,A -85,B 0,C 180,E1 -19618.29,E2 -19618.29} C_VEL
LIN {X 0,Y 235.568,Z 169.143,A -85,B 0,C 180,E1 -19621.71,E2 -19621.71} C_VEL
LIN {X 0,Y 235.344,Z 169.164,A -85,B 0,C 180,E1 -19626.861,E2 -19626.861} C_VEL
LIN {X 0,Y 235.177,Z 169.186,A -85,B 0,C 180,E1 -19630.329,E2 -19630.329} C_VEL
LIN {X 0,Y 235.05,Z 169.207,A -85,B 0,C 180,E1 -19635.611,E2 -19635.611} C_VEL
LIN {X 0,Y 234.954,Z 169.206,A -85,B 0,C 180,E1 -19639.21,E2 -19639.21} C_VEL
LIN {X 0,Y 234.925,Z 169.222,A -85,B 0,C 180,E1 -19642.887,E2 -19642.887} C_VEL
LIN {X 0,Y 234.923,Z 169.211,A -85,B 0,C 180,E1 -19646.663,E2 -19646.663} C_VEL
LIN {X 0,Y 234.893,Z 169.222,A -85,B 0,C 180,E1 -19650.574,E2 -19650.574} C_VEL
LIN {X 0,Y 234.92,Z 169.223,A -85,B 0,C 180,E1 -19654.64,E2 -19654.64} C_VEL
LIN {X 0,Y 234.907,Z 169.225,A -85,B 0,C 180,E1 -19658.936,E2 -19658.936} C_VEL
LIN {X 0,Y 234.859,Z 169.228,A -85,B 0,C 180,E1 -19663.493,E2 -19663.493} C_VEL
LIN {X 0,Y 234.872,Z 169.227,A -85,B 0,C 180,E1 -19666.513,E2 -19666.513} C_VEL
LIN {X 0,Y 234.915,Z 169.22,A -85,B 0,C 180,E1 -19671.08,E2 -19671.08} C_VEL
LIN {X 0,Y 234.962,Z 169.265,A -85,B 0,C 180,E1 -19674.434,E2 -19674.434} C_VEL
LIN {X 0,Y 235.945,Z 172.066,A -85,B 0,C 180,E1 -19674.709,E2 -19674.709} C_VEL
LIN {X 0,Y 237.472,Z 174.278,A -85,B 0,C 180,E1 -19675.052,E2 -19675.052} C_VEL
LIN {X 0,Y 243.985,Z 185.863,A -85,B 0,C 180,E1 -19676.528,E2 -19676.528} C_VEL
LIN {X 0,Y 250.329,Z 199.389,A -85,B 0,C 180,E1 -19677.944,E2 -19677.944} C_VEL
LIN {X 0,Y 255.144,Z 211.368,A -85,B 0,C 180,E1 -19679.013,E2 -19679.013} C_VEL
LIN {X 0,Y 252.763,Z 274.939,A -85,B 0,C 180,E1 -19680.781,E2 -19680.781} C_VEL
LIN {X 0,Y 251.796,Z 287.528,A -85,B 0,C 180,E1 -19681.408,E2 -19681.408} C_VEL
LIN {X 0,Y 250.419,Z 299.656,A -85,B 0,C 180,E1 -19682.302,E2 -19682.302} C_VEL
LIN {X 0,Y 248.569,Z 312.085,A -85,B 0,C 180,E1 -19683.558,E2 -19683.558} C_VEL
LIN {X 0,Y 246.386,Z 323.712,A -85,B 0,C 180,E1 -19685.12,E2 -19685.12} C_VEL
LIN {X 0,Y 244.548,Z 332.721,A -85,B 0,C 180,E1 -19686.65,E2 -19686.65} C_VEL
LIN {X 0,Y 242.394,Z 342.664,A -85,B 0,C 180,E1 -19688.752,E2 -19688.752} C_VEL
LIN {X 0,Y 240.293,Z 350.521,A -85,B 0,C 180,E1 -19690.791,E2 -19690.791} C_VEL
LIN {X 0,Y 238.141,Z 358.194,A -85,B 0,C 180,E1 -19693.278,E2 -19693.278} C_VEL
LIN {X 0,Y 236.201,Z 365.234,A -85,B 0,C 180,E1 -19696.231,E2 -19696.231} C_VEL
LIN {X 0,Y 234.87,Z 369.921,A -85,B 0,C 180,E1 -19698.786,E2 -19698.786} C_VEL
LIN {X 0,Y 233.946,Z 373.503,A -85,B 0,C 180,E1 -19701.362,E2 -19701.362} C_VEL
LIN {X 0,Y 233.494,Z 375.586,A -85,B 0,C 180,E1 -19703.355,E2 -19703.355} C_VEL
LIN {X 0,Y 233.065,Z 377.727,A -85,B 0,C 180,E1 -19706.543,E2 -19706.543} C_VEL
LIN {X 0,Y 232.947,Z 378.334,A -85,B 0,C 180,E1 -19708.272,E2 -19708.272} C_VEL
LIN {X 0,Y 232.902,Z 378.563,A -85,B 0,C 180,E1 -19710.001,E2 -19710.001} C_VEL
LIN {X 0,Y 232.947,Z 378.37,A -85,B 0,C 180,E1 -19711.73,E2 -19711.73} C_VEL
LIN {X 0,Y 233.063,Z 377.786,A -85,B 0,C 180,E1 -19713.458,E2 -19713.458} C_VEL
LIN {X 0,Y 233.544,Z 375.468,A -85,B 0,C 180,E1 -19716.914,E2 -19716.914} C_VEL
LIN {X 0,Y 234.196,Z 372.608,A -85,B 0,C 180,E1 -19719.501,E2 -19719.501} C_VEL
LIN {X 0,Y 235.229,Z 368.725,A -85,B 0,C 180,E1 -19722.073,E2 -19722.073} C_VEL
LIN {X 0,Y 236.66,Z 363.711,A -85,B 0,C 180,E1 -19724.622,E2 -19724.622} C_VEL
LIN {X 0,Y 238.36,Z 357.399,A -85,B 0,C 180,E1 -19727.149,E2 -19727.149} C_VEL
LIN {X 0,Y 240.621,Z 349.489,A -85,B 0,C 180,E1 -19729.627,E2 -19729.627} C_VEL
LIN {X 0,Y 242.691,Z 341.427,A -85,B 0,C 180,E1 -19731.668,E2 -19731.668} C_VEL
LIN {X 0,Y 244.833,Z 331.594,A -85,B 0,C 180,E1 -19733.696,E2 -19733.696} C_VEL
LIN {X 0,Y 247.173,Z 320.509,A -85,B 0,C 180,E1 -19735.472,E2 -19735.472} C_VEL
LIN {X 0,Y 249.114,Z 309.641,A -85,B 0,C 180,E1 -19736.834,E2 -19736.834} C_VEL
LIN {X 0,Y 250.79,Z 297.628,A -85,B 0,C 180,E1 -19737.995,E2 -19737.995} C_VEL
LIN {X 0,Y 252.118,Z 285.261,A -85,B 0,C 180,E1 -19738.856,E2 -19738.856} C_VEL
LIN {X 0,Y 253.037,Z 272.406,A -85,B 0,C 180,E1 -19739.424,E2 -19739.424} C_VEL
LIN {X 0,Y 255.224,Z 211.485,A -85,B 0,C 180,E1 -19741.111,E2 -19741.111} C_VEL
LIN {X 0,Y 249.131,Z 196.611,A -85,B 0,C 180,E1 -19742.466,E2 -19742.466} C_VEL
LIN {X 0,Y 242.414,Z 182.797,A -85,B 0,C 180,E1 -19743.975,E2 -19743.975} C_VEL
LIN {X 0,Y 236.517,Z 172.876,A -85,B 0,C 180,E1 -19745.314,E2 -19745.314} C_VEL
LIN {X 0,Y 235.076,Z 170.026,A -85,B 0,C 180,E1 -19745.67,E2 -19745.67} C_VEL
LIN {X 0,Y 234.943,Z 169.22,A -85,B 0,C 180,E1 -19745.794,E2 -19745.794} C_VEL
LIN {X 0,Y 234.913,Z 169.22,A -85,B 0,C 180,E1 -19748.935,E2 -19748.935} C_VEL
LIN {X 0,Y 234.853,Z 169.232,A -85,B 0,C 180,E1 -19753.494,E2 -19753.494} C_VEL
LIN {X 0,Y 234.854,Z 169.226,A -85,B 0,C 180,E1 -19756.506,E2 -19756.506} C_VEL
LIN {X 0,Y 234.919,Z 169.216,A -85,B 0,C 180,E1 -19761.079,E2 -19761.079} C_VEL
LIN {X 0,Y 234.926,Z 169.211,A -85,B 0,C 180,E1 -19765.361,E2 -19765.361} C_VEL
LIN {X 0,Y 234.9,Z 169.218,A -85,B 0,C 180,E1 -19769.427,E2 -19769.427} C_VEL
LIN {X 0,Y 234.97,Z 169.215,A -85,B 0,C 180,E1 -19773.807,E2 -19773.807} C_VEL
LIN {X 0,Y 234.969,Z 169.208,A -85,B 0,C 180,E1 -19778.966,E2 -19778.966} C_VEL
LIN {X 0,Y 235.05,Z 169.198,A -85,B 0,C 180,E1 -19783.097,E2 -19783.097} C_VEL
LIN {X 0,Y 235.091,Z 169.198,A -85,B 0,C 180,E1 -19787.921,E2 -19787.921} C_VEL
LIN {X 0,Y 235.311,Z 169.165,A -85,B 0,C 180,E1 -19791.412,E2 -19791.412} C_VEL
LIN {X 0,Y 235.346,Z 169.15,A -85,B 0,C 180,E1 -19793.14,E2 -19793.14} C_VEL
LIN {X 0,Y 235.574,Z 169.138,A -85,B 0,C 180,E1 -19798.29,E2 -19798.29} C_VEL
LIN {X 0,Y 235.572,Z 169.122,A -85,B 0,C 180,E1 -19801.71,E2 -19801.71} C_VEL
LIN {X 0,Y 235.34,Z 169.166,A -85,B 0,C 180,E1 -19806.86,E2 -19806.86} C_VEL
LIN {X 0,Y 235.183,Z 169.176,A -85,B 0,C 180,E1 -19810.329,E2 -19810.329} C_VEL
LIN {X 0,Y 235.039,Z 169.194,A -85,B 0,C 180,E1 -19815.611,E2 -19815.611} C_VEL
LIN {X 0,Y 234.939,Z 169.216,A -85,B 0,C 180,E1 -19819.43,E2 -19819.43} C_VEL
LIN {X 0,Y 234.233,Z 169.307,A -85,B 0,C 180,E1 -19820.859,E2 -19820.859} C_VEL
LIN {X 0,Y 231.416,Z 169.657,A -85,B 0,C 180,E1 -19823.193,E2 -19823.193} C_VEL
LIN {X 0,Y 228.215,Z 170.057,A -85,B 0,C 180,E1 -19826.073,E2 -19826.073} C_VEL
LIN {X 0,Y 227.866,Z 170.097,A -85,B 0,C 180,E1 -19827.07,E2 -19827.07} C_VEL
LIN {X 0,Y 227.856,Z 170.102,A -85,B 0,C 180,E1 -19831.624,E2 -19831.624} C_VEL
LIN {X 0,Y 227.865,Z 170.101,A -85,B 0,C 180,E1 -19835.875,E2 -19835.875} C_VEL
LIN {X 0,Y 227.801,Z 170.11,A -85,B 0,C 180,E1 -19840.382,E2 -19840.382} C_VEL
LIN {X 0,Y 227.811,Z 170.104,A -85,B 0,C 180,E1 -19845.199,E2 -19845.199} C_VEL
LIN {X 0,Y 227.815,Z 170.273,A -85,B 0,C 180,E1 -19848.055,E2 -19848.055} C_VEL
LIN {X 0,Y 230.054,Z 178.3,A -85,B 0,C 180,E1 -19851.972,E2 -19851.972} C_VEL
LIN {X 0,Y 230.949,Z 181.839,A -85,B 0,C 180,E1 -19853.564,E2 -19853.564} C_VEL
LIN {X 0,Y 239.394,Z 199.712,A -85,B 0,C 180,E1 -19855.666,E2 -19855.666} C_VEL
LIN {X 0,Y 244.791,Z 212.738,A -85,B 0,C 180,E1 -19856.964,E2 -19856.964} C_VEL
LIN {X 0,Y 248.033,Z 235.849,A -85,B 0,C 180,E1 -19858.217,E2 -19858.217} C_VEL
LIN {X 0,Y 247.995,Z 243.011,A -85,B 0,C 180,E1 -19858.45,E2 -19858.45} C_VEL
LIN {X 0,Y 246.104,Z 291.735,A -85,B 0,C 180,E1 -19859.864,E2 -19859.864} C_VEL
LIN {X 0,Y 244.807,Z 305.206,A -85,B 0,C 180,E1 -19860.557,E2 -19860.557} C_VEL
LIN {X 0,Y 243.05,Z 317.568,A -85,B 0,C 180,E1 -19861.503,E2 -19861.503} C_VEL
LIN {X 0,Y 241.06,Z 328.663,A -85,B 0,C 180,E1 -19862.665,E2 -19862.665} C_VEL
LIN {X 0,Y 238.622,Z 340.234,A -85,B 0,C 180,E1 -19864.251,E2 -19864.251} C_VEL
LIN {X 0,Y 236.128,Z 350.657,A -85,B 0,C 180,E1 -19866.075,E2 -19866.075} C_VEL
LIN {X 0,Y 233.935,Z 359.184,A -85,B 0,C 180,E1 -19867.942,E2 -19867.942} C_VEL
LIN {X 0,Y 231.911,Z 367.319,A -85,B 0,C 180,E1 -19870.149,E2 -19870.149} C_VEL
LIN {X 0,Y 229.819,Z 374.752,A -85,B 0,C 180,E1 -19872.652,E2 -19872.652} C_VEL
LIN {X 0,Y 228.416,Z 380.03,A -85,B 0,C 180,E1 -19874.838,E2 -19874.838} C_VEL
LIN {X 0,Y 227.062,Z 385.146,A -85,B 0,C 180,E1 -19877.486,E2 -19877.486} C_VEL
LIN {X 0,Y 226.266,Z 389.128,A -85,B 0,C 180,E1 -19880.163,E2 -19880.163} C_VEL
LIN {X 0,Y 225.768,Z 392.073,A -85,B 0,C 180,E1 -19882.846,E2 -19882.846} C_VEL
LIN {X 0,Y 225.604,Z 394.004,A -85,B 0,C 180,E1 -19885.463,E2 -19885.463} C_VEL
LIN {X 0,Y 225.703,Z 395.096,A -85,B 0,C 180,E1 -19888.215,E2 -19888.215} C_VEL
LIN {X 0,Y 225.795,Z 395.313,A -85,B 0,C 180,E1 -19889.999,E2 -19889.999} C_VEL
LIN {X 0,Y 225.703,Z 395.085,A -85,B 0,C 180,E1 -19891.783,E2 -19891.783} C_VEL
LIN {X 0,Y 225.643,Z 393.453,A -85,B 0,C 180,E1 -19895.36,E2 -19895.36} C_VEL
LIN {X 0,Y 225.773,Z 392.038,A -85,B 0,C 180,E1 -19897.152,E2 -19897.152} C_VEL
LIN {X 0,Y 226.278,Z 389.077,A -85,B 0,C 180,E1 -19899.835,E2 -19899.835} C_VEL
LIN {X 0,Y 227.06,Z 385.074,A -85,B 0,C 180,E1 -19902.512,E2 -19902.512} C_VEL
LIN {X 0,Y 228.663,Z 378.934,A -85,B 0,C 180,E1 -19905.6,E2 -19905.6} C_VEL
LIN {X 0,Y 230.509,Z 372.235,A -85,B 0,C 180,E1 -19908.209,E2 -19908.209} C_VEL
LIN {X 0,Y 232.795,Z 363.631,A -85,B 0,C 180,E1 -19910.866,E2 -19910.866} C_VEL
LIN {X 0,Y 234.871,Z 355.411,A -85,B 0,C 180,E1 -19912.891,E2 -19912.891} C_VEL
LIN {X 0,Y 237.445,Z 344.897,A -85,B 0,C 180,E1 -19914.945,E2 -19914.945} C_VEL
LIN {X 0,Y 240.096,Z 333.067,A -85,B 0,C 180,E1 -19916.746,E2 -19916.746} C_VEL
LIN {X 0,Y 242.367,Z 321.151,A -85,B 0,C 180,E1 -19918.111,E2 -19918.111} C_VEL
LIN {X 0,Y 244.256,Z 308.748,A -85,B 0,C 180,E1 -19919.165,E2 -19919.165} C_VEL
LIN {X 0,Y 245.709,Z 295.64,A -85,B 0,C 180,E1 -19919.935,E2 -19919.935} C_VEL
LIN {X 0,Y 246.474,Z 280.949,A -85,B 0,C 180,E1 -19920.453,E2 -19920.453} C_VEL
LIN {X 0,Y 248.079,Z 236.771,A -85,B 0,C 180,E1 -19921.694,E2 -19921.694} C_VEL
LIN {X 0,Y 244.683,Z 212.527,A -85,B 0,C 180,E1 -19923.006,E2 -19923.006} C_VEL
LIN {X 0,Y 238.176,Z 197.065,A -85,B 0,C 180,E1 -19924.569,E2 -19924.569} C_VEL
LIN {X 0,Y 232.37,Z 185.095,A -85,B 0,C 180,E1 -19925.996,E2 -19925.996} C_VEL
LIN {X 0,Y 230.845,Z 181.727,A -85,B 0,C 180,E1 -19926.401,E2 -19926.401} C_VEL
LIN {X 0,Y 228.969,Z 174.273,A -85,B 0,C 180,E1 -19929.883,E2 -19929.883} C_VEL
LIN {X 0,Y 227.789,Z 170.105,A -85,B 0,C 180,E1 -19931.972,E2 -19931.972} C_VEL
LIN {X 0,Y 227.806,Z 170.11,A -85,B 0,C 180,E1 -19935.198,E2 -19935.198} C_VEL
LIN {X 0,Y 227.795,Z 170.106,A -85,B 0,C 180,E1 -19939.617,E2 -19939.617} C_VEL
LIN {X 0,Y 227.86,Z 170.099,A -85,B 0,C 180,E1 -19944.124,E2 -19944.124} C_VEL
LIN {X 0,Y 227.85,Z 170.098,A -85,B 0,C 180,E1 -19948.375,E2 -19948.375} C_VEL
LIN {X 0,Y 227.839,Z 170.093,A -85,B 0,C 180,E1 -19952.439,E2 -19952.439} C_VEL
LIN {X 0,Y 227.859,Z 170.092,A -85,B 0,C 180,E1 -19956.361,E2 -19956.361} C_VEL
LIN {X 0,Y 227.881,Z 170.099,A -85,B 0,C 180,E1 -19960.169,E2 -19960.169} C_VEL
LIN {X 0,Y 227.992,Z 170.071,A -85,B 0,C 180,E1 -19963.893,E2 -19963.893} C_VEL
LIN {X 0,Y 228.117,Z 170.059,A -85,B 0,C 180,E1 -19969.348,E2 -19969.348} C_VEL
LIN {X 0,Y 228.285,Z 170.048,A -85,B 0,C 180,E1 -19972.926,E2 -19972.926} C_VEL
LIN {X 0,Y 228.523,Z 170.006,A -85,B 0,C 180,E1 -19978.238,E2 -19978.238} C_VEL
LIN {X 0,Y 228.526,Z 170.02,A -85,B 0,C 180,E1 -19981.762,E2 -19981.762} C_VEL
LIN {X 0,Y 228.297,Z 170.042,A -85,B 0,C 180,E1 -19987.073,E2 -19987.073} C_VEL
LIN {X 0,Y 228.118,Z 170.064,A -85,B 0,C 180,E1 -19990.653,E2 -19990.653} C_VEL
LIN {X 0,Y 228.001,Z 170.084,A -85,B 0,C 180,E1 -19996.106,E2 -19996.106} C_VEL
LIN {X 0,Y 227.918,Z 170.093,A -85,B 0,C 180,E1 -20001.718,E2 -20001.718} C_VEL
LIN {X 0,Y 227.9,Z 170.085,A -85,B 0,C 180,E1 -20006.585,E2 -20006.585} C_VEL
LIN {X 0,Y 227.868,Z 170.098,A -85,B 0,C 180,E1 -20010.281,E2 -20010.281} C_VEL
LIN {X 0,Y 227.871,Z 170.1,A -85,B 0,C 180,E1 -20013.722,E2 -20013.722} C_VEL
LIN {X 0,Y 227.835,Z 170.102,A -85,B 0,C 180,E1 -20018.093,E2 -20018.093} C_VEL
LIN {X 0,Y 227.787,Z 170.11,A -85,B 0,C 180,E1 -20022.748,E2 -20022.748} C_VEL
LIN {X 0,Y 227.818,Z 170.1,A -85,B 0,C 180,E1 -20025.197,E2 -20025.197} C_VEL
LIN {X 0,Y 227.806,Z 170.107,A -85,B 0,C 180,E1 -20029.621,E2 -20029.621} C_VEL
LIN {X 0,Y 227.88,Z 170.101,A -85,B 0,C 180,E1 -20033.142,E2 -20033.142} C_VEL
LIN {X 0,Y 228.88,Z 172.92,A -85,B 0,C 180,E1 -20033.466,E2 -20033.466} C_VEL
LIN {X 0,Y 230.651,Z 175.504,A -85,B 0,C 180,E1 -20033.893,E2 -20033.893} C_VEL
LIN {X 0,Y 238.333,Z 188.78,A -85,B 0,C 180,E1 -20035.719,E2 -20035.719} C_VEL
LIN {X 0,Y 244.481,Z 201.922,A -85,B 0,C 180,E1 -20037.159,E2 -20037.159} C_VEL
LIN {X 0,Y 249.057,Z 213.229,A -85,B 0,C 180,E1 -20038.221,E2 -20038.221} C_VEL
LIN {X 0,Y 246.579,Z 275.85,A -85,B 0,C 180,E1 -20040.007,E2 -20040.007} C_VEL
LIN {X 0,Y 245.446,Z 289.29,A -85,B 0,C 180,E1 -20040.713,E2 -20040.713} C_VEL
LIN {X 0,Y 244.03,Z 301.049,A -85,B 0,C 180,E1 -20041.629,E2 -20041.629} C_VEL
LIN {X 0,Y 242.258,Z 312.349,A -85,B 0,C 180,E1 -20042.813,E2 -20042.813} C_VEL
LIN {X 0,Y 239.965,Z 323.975,A -85,B 0,C 180,E1 -20044.407,E2 -20044.407} C_VEL
LIN {X 0,Y 238.015,Z 333.145,A -85,B 0,C 180,E1 -20046.004,E2 -20046.004} C_VEL
LIN {X 0,Y 235.789,Z 342.927,A -85,B 0,C 180,E1 -20048.127,E2 -20048.127} C_VEL
LIN {X 0,Y 233.605,Z 350.782,A -85,B 0,C 180,E1 -20050.218,E2 -20050.218} C_VEL
LIN {X 0,Y 231.351,Z 358.455,A -85,B 0,C 180,E1 -20052.773,E2 -20052.773} C_VEL
LIN {X 0,Y 229.32,Z 365.494,A -85,B 0,C 180,E1 -20055.809,E2 -20055.809} C_VEL
LIN {X 0,Y 227.915,Z 370.181,A -85,B 0,C 180,E1 -20058.439,E2 -20058.439} C_VEL
LIN {X 0,Y 226.918,Z 373.764,A -85,B 0,C 180,E1 -20061.093,E2 -20061.093} C_VEL
LIN {X 0,Y 226.397,Z 376.049,A -85,B 0,C 180,E1 -20063.4,E2 -20063.4} C_VEL
LIN {X 0,Y 225.991,Z 377.986,A -85,B 0,C 180,E1 -20066.435,E2 -20066.435} C_VEL
LIN {X 0,Y 225.835,Z 378.821,A -85,B 0,C 180,E1 -20070.001,E2 -20070.001} C_VEL
LIN {X 0,Y 225.861,Z 378.629,A -85,B 0,C 180,E1 -20071.784,E2 -20071.784} C_VEL
LIN {X 0,Y 225.989,Z 378.044,A -85,B 0,C 180,E1 -20073.567,E2 -20073.567} C_VEL
LIN {X 0,Y 226.499,Z 375.727,A -85,B 0,C 180,E1 -20077.131,E2 -20077.131} C_VEL
LIN {X 0,Y 227.196,Z 372.866,A -85,B 0,C 180,E1 -20079.796,E2 -20079.796} C_VEL
LIN {X 0,Y 228.281,Z 368.983,A -85,B 0,C 180,E1 -20082.446,E2 -20082.446} C_VEL
LIN {X 0,Y 229.804,Z 363.969,A -85,B 0,C 180,E1 -20085.068,E2 -20085.068} C_VEL
LIN {X 0,Y 231.589,Z 357.656,A -85,B 0,C 180,E1 -20087.667,E2 -20087.667} C_VEL
LIN {X 0,Y 233.934,Z 349.746,A -85,B 0,C 180,E1 -20090.212,E2 -20090.212} C_VEL
LIN {X 0,Y 236.099,Z 341.684,A -85,B 0,C 180,E1 -20092.305,E2 -20092.305} C_VEL
LIN {X 0,Y 238.352,Z 331.849,A -85,B 0,C 180,E1 -20094.381,E2 -20094.381} C_VEL
LIN {X 0,Y 240.802,Z 320.763,A -85,B 0,C 180,E1 -20096.196,E2 -20096.196} C_VEL
LIN {X 0,Y 242.822,Z 309.893,A -85,B 0,C 180,E1 -20097.587,E2 -20097.587} C_VEL
LIN {X 0,Y 244.548,Z 297.879,A -85,B 0,C 180,E1 -20098.776,E2 -20098.776} C_VEL
LIN {X 0,Y 245.982,Z 284.852,A -85,B 0,C 180,E1 -20099.689,E2 -20099.689} C_VEL
LIN {X 0,Y 246.936,Z 272.002,A -85,B 0,C 180,E1 -20100.251,E2 -20100.251} C_VEL
LIN {X 0,Y 249.081,Z 213.091,A -85,B 0,C 180,E1 -20101.922,E2 -20101.922} C_VEL
LIN {X 0,Y 242.255,Z 196.835,A -85,B 0,C 180,E1 -20103.509,E2 -20103.509} C_VEL
LIN {X 0,Y 236.25,Z 184.856,A -85,B 0,C 180,E1 -20104.922,E2 -20104.922} C_VEL
LIN {X 0,Y 229.699,Z 174.037,A -85,B 0,C 180,E1 -20106.494,E2 -20106.494} C_VEL
LIN {X 0,Y 228.158,Z 171.429,A -85,B 0,C 180,E1 -20106.884,E2 -20106.884} C_VEL
LIN {X 0,Y 227.874,Z 170.097,A -85,B 0,C 180,E1 -20107.023,E2 -20107.023} C_VEL
LIN {X 0,Y 227.799,Z 170.11,A -85,B 0,C 180,E1 -20110.383,E2 -20110.383} C_VEL
LIN {X 0,Y 227.811,Z 170.102,A -85,B 0,C 180,E1 -20115.199,E2 -20115.199} C_VEL
LIN {X 0,Y 227.802,Z 170.098,A -85,B 0,C 180,E1 -20119.618,E2 -20119.618} C_VEL
LIN {X 0,Y 227.866,Z 170.092,A -85,B 0,C 180,E1 -20124.125,E2 -20124.125} C_VEL
LIN {X 0,Y 227.857,Z 170.102,A -85,B 0,C 180,E1 -20128.375,E2 -20128.375} C_VEL
LIN {X 0,Y 227.856,Z 170.096,A -85,B 0,C 180,E1 -20132.441,E2 -20132.441} C_VEL
LIN {X 0,Y 227.895,Z 170.086,A -85,B 0,C 180,E1 -20136.365,E2 -20136.365} C_VEL
LIN {X 0,Y 227.912,Z 170.093,A -85,B 0,C 180,E1 -20140.172,E2 -20140.172} C_VEL
LIN {X 0,Y 228,Z 170.071,A -85,B 0,C 180,E1 -20143.894,E2 -20143.894} C_VEL
LIN {X 0,Y 228.141,Z 170.066,A -85,B 0,C 180,E1 -20149.348,E2 -20149.348} C_VEL
LIN {X 0,Y 228.299,Z 170.027,A -85,B 0,C 180,E1 -20152.927,E2 -20152.927} C_VEL
LIN {X 0,Y 228.533,Z 170.015,A -85,B 0,C 180,E1 -20158.238,E2 -20158.238} C_VEL
LIN {X 0,Y 228.53,Z 169.998,A -85,B 0,C 180,E1 -20161.762,E2 -20161.762} C_VEL
LIN {X 0,Y 228.292,Z 170.044,A -85,B 0,C 180,E1 -20167.073,E2 -20167.073} C_VEL
LIN {X 0,Y 228.124,Z 170.057,A -85,B 0,C 180,E1 -20170.652,E2 -20170.652} C_VEL
LIN {X 0,Y 227.998,Z 170.067,A -85,B 0,C 180,E1 -20176.106,E2 -20176.106} C_VEL
LIN {X 0,Y 227.918,Z 170.088,A -85,B 0,C 180,E1 -20181.717,E2 -20181.717} C_VEL
LIN {X 0,Y 227.866,Z 170.097,A -85,B 0,C 180,E1 -20187.07,E2 -20187.07} C_VEL
LIN {X 0,Y 227.142,Z 170.186,A -85,B 0,C 180,E1 -20188.544,E2 -20188.544} C_VEL
LIN {X 0,Y 224.271,Z 170.547,A -85,B 0,C 180,E1 -20190.95,E2 -20190.95} C_VEL
LIN {X 0,Y 221.876,Z 170.841,A -85,B 0,C 180,E1 -20192.913,E2 -20192.913} C_VEL
LIN {X 0,Y 220.868,Z 170.964,A -85,B 0,C 180,E1 -20194.437,E2 -20194.437} C_VEL
LIN {X 0,Y 220.794,Z 170.976,A -85,B 0,C 180,E1 -20194.953,E2 -20194.953} C_VEL
LIN {X 0,Y 220.8,Z 170.975,A -85,B 0,C 180,E1 -20197.274,E2 -20197.274} C_VEL
LIN {X 0,Y 220.748,Z 170.982,A -85,B 0,C 180,E1 -20201.958,E2 -20201.958} C_VEL
LIN {X 0,Y 220.739,Z 170.987,A -85,B 0,C 180,E1 -20206.388,E2 -20206.388} C_VEL
LIN {X 0,Y 220.756,Z 171.107,A -85,B 0,C 180,E1 -20206.941,E2 -20206.941} C_VEL
LIN {X 0,Y 222.935,Z 178.846,A -85,B 0,C 180,E1 -20210.913,E2 -20210.913} C_VEL
LIN {X 0,Y 223.567,Z 181.402,A -85,B 0,C 180,E1 -20212.148,E2 -20212.148} C_VEL
LIN {X 0,Y 225.6,Z 185.527,A -85,B 0,C 180,E1 -20212.707,E2 -20212.707} C_VEL
LIN {X 0,Y 232.24,Z 199.112,A -85,B 0,C 180,E1 -20214.44,E2 -20214.44} C_VEL
LIN {X 0,Y 238.909,Z 214.896,A -85,B 0,C 180,E1 -20216.126,E2 -20216.126} C_VEL
LIN {X 0,Y 241.644,Z 234.112,A -85,B 0,C 180,E1 -20217.223,E2 -20217.223} C_VEL
LIN {X 0,Y 242.131,Z 239.839,A -85,B 0,C 180,E1 -20217.493,E2 -20217.493} C_VEL
LIN {X 0,Y 240.033,Z 290.915,A -85,B 0,C 180,E1 -20218.988,E2 -20218.988} C_VEL
LIN {X 0,Y 238.739,Z 304.301,A -85,B 0,C 180,E1 -20219.679,E2 -20219.679} C_VEL
LIN {X 0,Y 236.828,Z 317.314,A -85,B 0,C 180,E1 -20220.682,E2 -20220.682} C_VEL
LIN {X 0,Y 234.428,Z 329.993,A -85,B 0,C 180,E1 -20222.067,E2 -20222.067} C_VEL
LIN {X 0,Y 231.938,Z 341.273,A -85,B 0,C 180,E1 -20223.694,E2 -20223.694} C_VEL
LIN {X 0,Y 229.363,Z 351.437,A -85,B 0,C 180,E1 -20225.565,E2 -20225.565} C_VEL
LIN {X 0,Y 226.89,Z 360.599,A -85,B 0,C 180,E1 -20227.7,E2 -20227.7} C_VEL
LIN {X 0,Y 224.526,Z 369.543,A -85,B 0,C 180,E1 -20230.336,E2 -20230.336} C_VEL
LIN {X 0,Y 222.465,Z 376.738,A -85,B 0,C 180,E1 -20233.008,E2 -20233.008} C_VEL
LIN {X 0,Y 220.977,Z 381.595,A -85,B 0,C 180,E1 -20235.259,E2 -20235.259} C_VEL
LIN {X 0,Y 219.772,Z 386.326,A -85,B 0,C 180,E1 -20238.002,E2 -20238.002} C_VEL
LIN {X 0,Y 219.018,Z 389.946,A -85,B 0,C 180,E1 -20240.767,E2 -20240.767} C_VEL
LIN {X 0,Y 218.691,Z 391.813,A -85,B 0,C 180,E1 -20242.614,E2 -20242.614} C_VEL
LIN {X 0,Y 218.52,Z 393.892,A -85,B 0,C 180,E1 -20245.573,E2 -20245.573} C_VEL
LIN {X 0,Y 218.616,Z 394.838,A -85,B 0,C 180,E1 -20248.157,E2 -20248.157} C_VEL
LIN {X 0,Y 218.706,Z 395.054,A -85,B 0,C 180,E1 -20249.999,E2 -20249.999} C_VEL
LIN {X 0,Y 218.615,Z 394.826,A -85,B 0,C 180,E1 -20251.841,E2 -20251.841} C_VEL
LIN {X 0,Y 218.564,Z 393.193,A -85,B 0,C 180,E1 -20255.535,E2 -20255.535} C_VEL
LIN {X 0,Y 218.7,Z 391.777,A -85,B 0,C 180,E1 -20257.384,E2 -20257.384} C_VEL
LIN {X 0,Y 219.267,Z 388.817,A -85,B 0,C 180,E1 -20260.152,E2 -20260.152} C_VEL
LIN {X 0,Y 220.084,Z 384.812,A -85,B 0,C 180,E1 -20262.915,E2 -20262.915} C_VEL
LIN {X 0,Y 221.813,Z 378.673,A -85,B 0,C 180,E1 -20266.094,E2 -20266.094} C_VEL
LIN {X 0,Y 223.767,Z 371.974,A -85,B 0,C 180,E1 -20268.778,E2 -20268.778} C_VEL
LIN {X 0,Y 226.08,Z 363.548,A -85,B 0,C 180,E1 -20271.46,E2 -20271.46} C_VEL
LIN {X 0,Y 228.313,Z 355.147,A -85,B 0,C 180,E1 -20273.587,E2 -20273.587} C_VEL
LIN {X 0,Y 231.029,Z 344.634,A -85,B 0,C 180,E1 -20275.688,E2 -20275.688} C_VEL
LIN {X 0,Y 233.761,Z 332.803,A -85,B 0,C 180,E1 -20277.531,E2 -20277.531} C_VEL
LIN {X 0,Y 236.129,Z 320.885,A -85,B 0,C 180,E1 -20278.923,E2 -20278.923} C_VEL
LIN {X 0,Y 238.092,Z 308.481,A -85,B 0,C 180,E1 -20279.996,E2 -20279.996} C_VEL
LIN {X 0,Y 239.557,Z 295.728,A -85,B 0,C 180,E1 -20280.765,E2 -20280.765} C_VEL
LIN {X 0,Y 240.336,Z 281.761,A -85,B 0,C 180,E1 -20281.279,E2 -20281.279} C_VEL
LIN {X 0,Y 241.976,Z 237.235,A -85,B 0,C 180,E1 -20282.565,E2 -20282.565} C_VEL
LIN {X 0,Y 238.964,Z 215.198,A -85,B 0,C 180,E1 -20283.797,E2 -20283.797} C_VEL
LIN {X 0,Y 232.714,Z 200.264,A -85,B 0,C 180,E1 -20285.373,E2 -20285.373} C_VEL
LIN {X 0,Y 227.2,Z 188.853,A -85,B 0,C 180,E1 -20286.794,E2 -20286.794} C_VEL
LIN {X 0,Y 224.845,Z 184.289,A -85,B 0,C 180,E1 -20287.419,E2 -20287.419} C_VEL
LIN {X 0,Y 223.568,Z 181.241,A -85,B 0,C 180,E1 -20287.855,E2 -20287.855} C_VEL
LIN {X 0,Y 221.147,Z 172.561,A -85,B 0,C 180,E1 -20292.219,E2 -20292.219} C_VEL
LIN {X 0,Y 220.744,Z 170.988,A -85,B 0,C 180,E1 -20293.083,E2 -20293.083} C_VEL
LIN {X 0,Y 220.739,Z 170.986,A -85,B 0,C 180,E1 -20297.076,E2 -20297.076} C_VEL
LIN {X 0,Y 220.776,Z 170.982,A -85,B 0,C 180,E1 -20300.457,E2 -20300.457} C_VEL
LIN {X 0,Y 220.82,Z 170.972,A -85,B 0,C 180,E1 -20302.792,E2 -20302.792} C_VEL
LIN {X 0,Y 220.806,Z 170.971,A -85,B 0,C 180,E1 -20307.242,E2 -20307.242} C_VEL
LIN {X 0,Y 220.793,Z 170.968,A -85,B 0,C 180,E1 -20311.48,E2 -20311.48} C_VEL
LIN {X 0,Y 220.796,Z 170.977,A -85,B 0,C 180,E1 -20315.557,E2 -20315.557} C_VEL
LIN {X 0,Y 220.839,Z 170.975,A -85,B 0,C 180,E1 -20319.509,E2 -20319.509} C_VEL
LIN {X 0,Y 220.959,Z 170.946,A -85,B 0,C 180,E1 -20323.366,E2 -20323.366} C_VEL
LIN {X 0,Y 221.042,Z 170.942,A -85,B 0,C 180,E1 -20329.002,E2 -20329.002} C_VEL
LIN {X 0,Y 221.222,Z 170.928,A -85,B 0,C 180,E1 -20332.699,E2 -20332.699} C_VEL
LIN {X 0,Y 221.456,Z 170.884,A -85,B 0,C 180,E1 -20338.181,E2 -20338.181} C_VEL
LIN {X 0,Y 221.459,Z 170.899,A -85,B 0,C 180,E1 -20341.819,E2 -20341.819} C_VEL
LIN {X 0,Y 221.234,Z 170.922,A -85,B 0,C 180,E1 -20347.3,E2 -20347.3} C_VEL
LIN {X 0,Y 221.04,Z 170.942,A -85,B 0,C 180,E1 -20350.998,E2 -20350.998} C_VEL
LIN {X 0,Y 220.963,Z 170.96,A -85,B 0,C 180,E1 -20356.634,E2 -20356.634} C_VEL
LIN {X 0,Y 220.843,Z 170.965,A -85,B 0,C 180,E1 -20360.491,E2 -20360.491} C_VEL
LIN {X 0,Y 220.825,Z 170.974,A -85,B 0,C 180,E1 -20364.44,E2 -20364.44} C_VEL
LIN {X 0,Y 220.795,Z 170.981,A -85,B 0,C 180,E1 -20368.52,E2 -20368.52} C_VEL
LIN {X 0,Y 220.807,Z 170.973,A -85,B 0,C 180,E1 -20372.758,E2 -20372.758} C_VEL
LIN {X 0,Y 220.797,Z 170.98,A -85,B 0,C 180,E1 -20377.276,E2 -20377.276} C_VEL
LIN {X 0,Y 220.747,Z 170.986,A -85,B 0,C 180,E1 -20381.958,E2 -20381.958} C_VEL
LIN {X 0,Y 220.76,Z 170.979,A -85,B 0,C 180,E1 -20385.545,E2 -20385.545} C_VEL
LIN {X 0,Y 220.782,Z 170.984,A -85,B 0,C 180,E1 -20390.46,E2 -20390.46} C_VEL
LIN {X 0,Y 220.801,Z 170.98,A -85,B 0,C 180,E1 -20391.802,E2 -20391.802} C_VEL
LIN {X 0,Y 221.827,Z 173.877,A -85,B 0,C 180,E1 -20392.129,E2 -20392.129} C_VEL
LIN {X 0,Y 223.51,Z 176.138,A -85,B 0,C 180,E1 -20392.557,E2 -20392.557} C_VEL
LIN {X 0,Y 231.664,Z 189.744,A -85,B 0,C 180,E1 -20394.611,E2 -20394.611} C_VEL
LIN {X 0,Y 238.128,Z 203.147,A -85,B 0,C 180,E1 -20396.199,E2 -20396.199} C_VEL
LIN {X 0,Y 243.004,Z 215.123,A -85,B 0,C 180,E1 -20397.388,E2 -20397.388} C_VEL
LIN {X 0,Y 240.496,Z 275.762,A -85,B 0,C 180,E1 -20399.148,E2 -20399.148} C_VEL
LIN {X 0,Y 239.385,Z 288.957,A -85,B 0,C 180,E1 -20399.848,E2 -20399.848} C_VEL
LIN {X 0,Y 237.809,Z 301.315,A -85,B 0,C 180,E1 -20400.817,E2 -20400.817} C_VEL
LIN {X 0,Y 235.987,Z 312.613,A -85,B 0,C 180,E1 -20402.028,E2 -20402.028} C_VEL
LIN {X 0,Y 233.586,Z 324.238,A -85,B 0,C 180,E1 -20403.656,E2 -20403.656} C_VEL
LIN {X 0,Y 231.284,Z 334.614,A -85,B 0,C 180,E1 -20405.531,E2 -20405.531} C_VEL
LIN {X 0,Y 229.216,Z 343.189,A -85,B 0,C 180,E1 -20407.465,E2 -20407.465} C_VEL
LIN {X 0,Y 226.942,Z 351.044,A -85,B 0,C 180,E1 -20409.612,E2 -20409.612} C_VEL
LIN {X 0,Y 224.558,Z 358.717,A -85,B 0,C 180,E1 -20412.234,E2 -20412.234} C_VEL
LIN {X 0,Y 222.439,Z 365.755,A -85,B 0,C 180,E1 -20415.36,E2 -20415.36} C_VEL
LIN {X 0,Y 220.979,Z 370.441,A -85,B 0,C 180,E1 -20418.071,E2 -20418.071} C_VEL
LIN {X 0,Y 219.919,Z 374.023,A -85,B 0,C 180,E1 -20420.807,E2 -20420.807} C_VEL
LIN {X 0,Y 219.293,Z 376.527,A -85,B 0,C 180,E1 -20423.466,E2 -20423.466} C_VEL
LIN {X 0,Y 218.92,Z 378.245,A -85,B 0,C 180,E1 -20426.32,E2 -20426.32} C_VEL
LIN {X 0,Y 218.747,Z 379.08,A -85,B 0,C 180,E1 -20430.001,E2 -20430.001} C_VEL
LIN {X 0,Y 218.777,Z 378.887,A -85,B 0,C 180,E1 -20431.842,E2 -20431.842} C_VEL
LIN {X 0,Y 218.917,Z 378.302,A -85,B 0,C 180,E1 -20433.682,E2 -20433.682} C_VEL
LIN {X 0,Y 219.468,Z 375.985,A -85,B 0,C 180,E1 -20437.36,E2 -20437.36} C_VEL
LIN {X 0,Y 220.196,Z 373.125,A -85,B 0,C 180,E1 -20440.111,E2 -20440.111} C_VEL
LIN {X 0,Y 221.353,Z 369.241,A -85,B 0,C 180,E1 -20442.842,E2 -20442.842} C_VEL
LIN {X 0,Y 222.945,Z 364.227,A -85,B 0,C 180,E1 -20445.543,E2 -20445.543} C_VEL
LIN {X 0,Y 224.84,Z 357.913,A -85,B 0,C 180,E1 -20448.215,E2 -20448.215} C_VEL
LIN {X 0,Y 227.285,Z 350.003,A -85,B 0,C 180,E1 -20450.831,E2 -20450.831} C_VEL
LIN {X 0,Y 229.54,Z 341.94,A -85,B 0,C 180,E1 -20452.978,E2 -20452.978} C_VEL
LIN {X 0,Y 231.921,Z 332.104,A -85,B 0,C 180,E1 -20455.104,E2 -20455.104} C_VEL
LIN {X 0,Y 234.473,Z 321.017,A -85,B 0,C 180,E1 -20456.959,E2 -20456.959} C_VEL
LIN {X 0,Y 236.566,Z 310.146,A -85,B 0,C 180,E1 -20458.382,E2 -20458.382} C_VEL
LIN {X 0,Y 238.376,Z 298.13,A -85,B 0,C 180,E1 -20459.594,E2 -20459.594} C_VEL
LIN {X 0,Y 239.82,Z 285.413,A -85,B 0,C 180,E1 -20460.511,E2 -20460.511} C_VEL
LIN {X 0,Y 240.878,Z 271.899,A -85,B 0,C 180,E1 -20461.109,E2 -20461.109} C_VEL
LIN {X 0,Y 243.088,Z 215.113,A -85,B 0,C 180,E1 -20462.745,E2 -20462.745} C_VEL
LIN {X 0,Y 236.598,Z 199.667,A -85,B 0,C 180,E1 -20464.326,E2 -20464.326} C_VEL
LIN {X 0,Y 231.346,Z 189.152,A -85,B 0,C 180,E1 -20465.621,E2 -20465.621} C_VEL
LIN {X 0,Y 224.858,Z 178.418,A -85,B 0,C 180,E1 -20467.247,E2 -20467.247} C_VEL
LIN {X 0,Y 222.685,Z 174.982,A -85,B 0,C 180,E1 -20467.815,E2 -20467.815} C_VEL
LIN {X 0,Y 221.135,Z 172.416,A -85,B 0,C 180,E1 -20468.234,E2 -20468.234} C_VEL
LIN {X 0,Y 220.782,Z 170.982,A -85,B 0,C 180,E1 -20468.422,E2 -20468.422} C_VEL
LIN {X 0,Y 220.744,Z 170.988,A -85,B 0,C 180,E1 -20472.923,E2 -20472.923} C_VEL
LIN {X 0,Y 220.745,Z 170.985,A -85,B 0,C 180,E1 -20477.077,E2 -20477.077} C_VEL
LIN {X 0,Y 220.782,Z 170.973,A -85,B 0,C 180,E1 -20480.458,E2 -20480.458} C_VEL
LIN {X 0,Y 220.826,Z 170.978,A -85,B 0,C 180,E1 -20482.793,E2 -20482.793} C_VEL
LIN {X 0,Y 220.813,Z 170.979,A -85,B 0,C 180,E1 -20487.243,E2 -20487.243} C_VEL
LIN {X 0,Y 220.805,Z 170.969,A -85,B 0,C 180,E1 -20491.482,E2 -20491.482} C_VEL
LIN {X 0,Y 220.848,Z 170.97,A -85,B 0,C 180,E1 -20495.563,E2 -20495.563} C_VEL
LIN {X 0,Y 220.87,Z 170.969,A -85,B 0,C 180,E1 -20499.512,E2 -20499.512} C_VEL
LIN {X 0,Y 220.967,Z 170.951,A -85,B 0,C 180,E1 -20503.366,E2 -20503.366} C_VEL
LIN {X 0,Y 221.06,Z 170.948,A -85,B 0,C 180,E1 -20509.003,E2 -20509.003} C_VEL
LIN {X 0,Y 221.237,Z 170.906,A -85,B 0,C 180,E1 -20512.7,E2 -20512.7} C_VEL
LIN {X 0,Y 221.466,Z 170.896,A -85,B 0,C 180,E1 -20518.181,E2 -20518.181} C_VEL
LIN {X 0,Y 221.463,Z 170.878,A -85,B 0,C 180,E1 -20521.818,E2 -20521.818} C_VEL
LIN {X 0,Y 221.229,Z 170.92,A -85,B 0,C 180,E1 -20527.3,E2 -20527.3} C_VEL
LIN {X 0,Y 221.046,Z 170.941,A -85,B 0,C 180,E1 -20530.997,E2 -20530.997} C_VEL
LIN {X 0,Y 220.944,Z 170.944,A -85,B 0,C 180,E1 -20536.635,E2 -20536.635} C_VEL
LIN {X 0,Y 220.844,Z 170.974,A -85,B 0,C 180,E1 -20540.491,E2 -20540.491} C_VEL
LIN {X 0,Y 220.796,Z 170.974,A -85,B 0,C 180,E1 -20544.443,E2 -20544.443} C_VEL
LIN {X 0,Y 220.799,Z 170.971,A -85,B 0,C 180,E1 -20548.519,E2 -20548.519} C_VEL
LIN {X 0,Y 220.813,Z 170.975,A -85,B 0,C 180,E1 -20552.757,E2 -20552.757} C_VEL
LIN {X 0,Y 220.794,Z 170.976,A -85,B 0,C 180,E1 -20554.953,E2 -20554.953} C_VEL
LIN {X 0,Y 220.124,Z 171.067,A -85,B 0,C 180,E1 -20556.474,E2 -20556.474} C_VEL
LIN {X 0,Y 217.206,Z 171.425,A -85,B 0,C 180,E1 -20558.955,E2 -20558.955} C_VEL
LIN {X 0,Y 214.743,Z 171.731,A -85,B 0,C 180,E1 -20560.981,E2 -20560.981} C_VEL
LIN {X 0,Y 213.726,Z 171.86,A -85,B 0,C 180,E1 -20562.557,E2 -20562.557} C_VEL
LIN {X 0,Y 213.665,Z 171.863,A -85,B 0,C 180,E1 -20563.091,E2 -20563.091} C_VEL
LIN {X 0,Y 213.723,Z 172.033,A -85,B 0,C 180,E1 -20565.785,E2 -20565.785} C_VEL
LIN {X 0,Y 216.277,Z 181.156,A -85,B 0,C 180,E1 -20570.635,E2 -20570.635} C_VEL
LIN {X 0,Y 218.546,Z 185.419,A -85,B 0,C 180,E1 -20571.293,E2 -20571.293} C_VEL
LIN {X 0,Y 225.66,Z 199.819,A -85,B 0,C 180,E1 -20573.275,E2 -20573.275} C_VEL
LIN {X 0,Y 231.707,Z 213.641,A -85,B 0,C 180,E1 -20574.886,E2 -20574.886} C_VEL
LIN {X 0,Y 233.423,Z 218.122,A -85,B 0,C 180,E1 -20575.343,E2 -20575.343} C_VEL
LIN {X 0,Y 236.099,Z 238.67,A -85,B 0,C 180,E1 -20576.522,E2 -20576.522} C_VEL
LIN {X 0,Y 234.027,Z 290.147,A -85,B 0,C 180,E1 -20578.071,E2 -20578.071} C_VEL
LIN {X 0,Y 232.72,Z 303.432,A -85,B 0,C 180,E1 -20578.757,E2 -20578.757} C_VEL
LIN {X 0,Y 230.826,Z 315.953,A -85,B 0,C 180,E1 -20579.716,E2 -20579.716} C_VEL
LIN {X 0,Y 228.536,Z 328.154,A -85,B 0,C 180,E1 -20581.03,E2 -20581.03} C_VEL
LIN {X 0,Y 225.893,Z 339.722,A -85,B 0,C 180,E1 -20582.683,E2 -20582.683} C_VEL
LIN {X 0,Y 223.215,Z 350.145,A -85,B 0,C 180,E1 -20584.596,E2 -20584.596} C_VEL
LIN {X 0,Y 220.796,Z 358.669,A -85,B 0,C 180,E1 -20586.554,E2 -20586.554} C_VEL
LIN {X 0,Y 218.204,Z 367.922,A -85,B 0,C 180,E1 -20589.249,E2 -20589.249} C_VEL
LIN {X 0,Y 215.899,Z 375.358,A -85,B 0,C 180,E1 -20591.985,E2 -20591.985} C_VEL
LIN {X 0,Y 214.101,Z 381.337,A -85,B 0,C 180,E1 -20594.775,E2 -20594.775} C_VEL
LIN {X 0,Y 212.796,Z 386.066,A -85,B 0,C 180,E1 -20597.603,E2 -20597.603} C_VEL
LIN {X 0,Y 212.003,Z 389.687,A -85,B 0,C 180,E1 -20600.458,E2 -20600.458} C_VEL
LIN {X 0,Y 211.631,Z 391.554,A -85,B 0,C 180,E1 -20602.366,E2 -20602.366} C_VEL
LIN {X 0,Y 211.42,Z 393.778,A -85,B 0,C 180,E1 -20605.758,E2 -20605.758} C_VEL
LIN {X 0,Y 211.51,Z 394.578,A -85,B 0,C 180,E1 -20608.095,E2 -20608.095} C_VEL
LIN {X 0,Y 211.619,Z 394.795,A -85,B 0,C 180,E1 -20609.999,E2 -20609.999} C_VEL
LIN {X 0,Y 211.51,Z 394.567,A -85,B 0,C 180,E1 -20611.903,E2 -20611.903} C_VEL
LIN {X 0,Y 211.419,Z 393.76,A -85,B 0,C 180,E1 -20614.24,E2 -20614.24} C_VEL
LIN {X 0,Y 211.64,Z 391.517,A -85,B 0,C 180,E1 -20617.632,E2 -20617.632} C_VEL
LIN {X 0,Y 212.234,Z 388.555,A -85,B 0,C 180,E1 -20620.493,E2 -20620.493} C_VEL
LIN {X 0,Y 213.125,Z 384.55,A -85,B 0,C 180,E1 -20623.345,E2 -20623.345} C_VEL
LIN {X 0,Y 214.989,Z 378.411,A -85,B 0,C 180,E1 -20626.62,E2 -20626.62} C_VEL
LIN {X 0,Y 217.049,Z 371.712,A -85,B 0,C 180,E1 -20629.382,E2 -20629.382} C_VEL
LIN {X 0,Y 219.374,Z 363.551,A -85,B 0,C 180,E1 -20632.062,E2 -20632.062} C_VEL
LIN {X 0,Y 221.791,Z 354.884,A -85,B 0,C 180,E1 -20634.325,E2 -20634.325} C_VEL
LIN {X 0,Y 224.641,Z 344.371,A -85,B 0,C 180,E1 -20636.474,E2 -20636.474} C_VEL
LIN {X 0,Y 227.474,Z 332.539,A -85,B 0,C 180,E1 -20638.359,E2 -20638.359} C_VEL
LIN {X 0,Y 229.935,Z 320.62,A -85,B 0,C 180,E1 -20639.779,E2 -20639.779} C_VEL
LIN {X 0,Y 231.984,Z 308.214,A -85,B 0,C 180,E1 -20640.871,E2 -20640.871} C_VEL
LIN {X 0,Y 233.563,Z 294.894,A -85,B 0,C 180,E1 -20641.678,E2 -20641.678} C_VEL
LIN {X 0,Y 234.39,Z 279.375,A -85,B 0,C 180,E1 -20642.241,E2 -20642.241} C_VEL
LIN {X 0,Y 235.992,Z 238.28,A -85,B 0,C 180,E1 -20643.451,E2 -20643.451} C_VEL
LIN {X 0,Y 233.208,Z 217.589,A -85,B 0,C 180,E1 -20644.652,E2 -20644.652} C_VEL
LIN {X 0,Y 226.503,Z 201.626,A -85,B 0,C 180,E1 -20646.432,E2 -20646.432} C_VEL
LIN {X 0,Y 218.52,Z 185.38,A -85,B 0,C 180,E1 -20648.641,E2 -20648.641} C_VEL
LIN {X 0,Y 216.197,Z 180.998,A -85,B 0,C 180,E1 -20649.344,E2 -20649.344} C_VEL
LIN {X 0,Y 213.711,Z 171.865,A -85,B 0,C 180,E1 -20654.297,E2 -20654.297} C_VEL
LIN {X 0,Y 213.698,Z 171.862,A -85,B 0,C 180,E1 -20659.146,E2 -20659.146} C_VEL
LIN {X 0,Y 213.736,Z 171.856,A -85,B 0,C 180,E1 -20663.71,E2 -20663.71} C_VEL
LIN {X 0,Y 213.753,Z 171.853,A -85,B 0,C 180,E1 -20668.26,E2 -20668.26} C_VEL
LIN {X 0,Y 213.778,Z 171.844,A -85,B 0,C 180,E1 -20672.597,E2 -20672.597} C_VEL
LIN {X 0,Y 213.788,Z 171.84,A -85,B 0,C 180,E1 -20676.989,E2 -20676.989} C_VEL
LIN {X 0,Y 213.871,Z 171.83,A -85,B 0,C 180,E1 -20682.798,E2 -20682.798} C_VEL
LIN {X 0,Y 213.903,Z 171.841,A -85,B 0,C 180,E1 -20686.703,E2 -20686.703} C_VEL
LIN {X 0,Y 214.116,Z 171.798,A -85,B 0,C 180,E1 -20690.554,E2 -20690.554} C_VEL
LIN {X 0,Y 214.059,Z 171.82,A -85,B 0,C 180,E1 -20694.347,E2 -20694.347} C_VEL
LIN {X 0,Y 214.393,Z 171.763,A -85,B 0,C 180,E1 -20698.122,E2 -20698.122} C_VEL
LIN {X 0,Y 214.504,Z 171.762,A -85,B 0,C 180,E1 -20700,E2 -20700} C_VEL
LIN {X 0,Y 214.396,Z 171.778,A -85,B 0,C 180,E1 -20701.879,E2 -20701.879} C_VEL
LIN {X 0,Y 214.175,Z 171.803,A -85,B 0,C 180,E1 -20707.542,E2 -20707.542} C_VEL
LIN {X 0,Y 213.972,Z 171.818,A -85,B 0,C 180,E1 -20711.366,E2 -20711.366} C_VEL
LIN {X 0,Y 213.864,Z 171.843,A -85,B 0,C 180,E1 -20715.242,E2 -20715.242} C_VEL
LIN {X 0,Y 213.785,Z 171.84,A -85,B 0,C 180,E1 -20719.193,E2 -20719.193} C_VEL
LIN {X 0,Y 213.784,Z 171.856,A -85,B 0,C 180,E1 -20723.234,E2 -20723.234} C_VEL
LIN {X 0,Y 213.779,Z 171.849,A -85,B 0,C 180,E1 -20727.428,E2 -20727.428} C_VEL
LIN {X 0,Y 213.754,Z 171.848,A -85,B 0,C 180,E1 -20731.74,E2 -20731.74} C_VEL
LIN {X 0,Y 213.737,Z 171.86,A -85,B 0,C 180,E1 -20736.29,E2 -20736.29} C_VEL
LIN {X 0,Y 213.695,Z 171.866,A -85,B 0,C 180,E1 -20741.13,E2 -20741.13} C_VEL
LIN {X 0,Y 213.698,Z 171.864,A -85,B 0,C 180,E1 -20743.681,E2 -20743.681} C_VEL
LIN {X 0,Y 213.699,Z 171.863,A -85,B 0,C 180,E1 -20746.346,E2 -20746.346} C_VEL
LIN {X 0,Y 213.762,Z 172.017,A -85,B 0,C 180,E1 -20750.33,E2 -20750.33} C_VEL
LIN {X 0,Y 214.83,Z 174.842,A -85,B 0,C 180,E1 -20750.689,E2 -20750.689} C_VEL
LIN {X 0,Y 216.557,Z 177.068,A -85,B 0,C 180,E1 -20751.159,E2 -20751.159} C_VEL
LIN {X 0,Y 224.88,Z 190.697,A -85,B 0,C 180,E1 -20753.398,E2 -20753.398} C_VEL
LIN {X 0,Y 229.654,Z 199.741,A -85,B 0,C 180,E1 -20754.628,E2 -20754.628} C_VEL
LIN {X 0,Y 235.359,Z 212.816,A -85,B 0,C 180,E1 -20756.092,E2 -20756.092} C_VEL
LIN {X 0,Y 236.943,Z 216.712,A -85,B 0,C 180,E1 -20756.491,E2 -20756.491} C_VEL
LIN {X 0,Y 234.706,Z 270.84,A -85,B 0,C 180,E1 -20758.07,E2 -20758.07} C_VEL
LIN {X 0,Y 233.743,Z 284.502,A -85,B 0,C 180,E1 -20758.675,E2 -20758.675} C_VEL
LIN {X 0,Y 232.285,Z 297.052,A -85,B 0,C 180,E1 -20759.552,E2 -20759.552} C_VEL
LIN {X 0,Y 230.403,Z 309.383,A -85,B 0,C 180,E1 -20760.789,E2 -20760.789} C_VEL
LIN {X 0,Y 228.185,Z 320.454,A -85,B 0,C 180,E1 -20762.237,E2 -20762.237} C_VEL
LIN {X 0,Y 225.567,Z 331.736,A -85,B 0,C 180,E1 -20764.14,E2 -20764.14} C_VEL
LIN {X 0,Y 223.191,Z 341.677,A -85,B 0,C 180,E1 -20766.331,E2 -20766.331} C_VEL
LIN {X 0,Y 220.731,Z 349.829,A -85,B 0,C 180,E1 -20768.523,E2 -20768.523} C_VEL
LIN {X 0,Y 218.188,Z 357.813,A -85,B 0,C 180,E1 -20771.211,E2 -20771.211} C_VEL
LIN {X 0,Y 216.145,Z 364.213,A -85,B 0,C 180,E1 -20773.957,E2 -20773.957} C_VEL
LIN {X 0,Y 214.491,Z 369.288,A -85,B 0,C 180,E1 -20776.742,E2 -20776.742} C_VEL
LIN {X 0,Y 213.248,Z 373.226,A -85,B 0,C 180,E1 -20779.558,E2 -20779.558} C_VEL
LIN {X 0,Y 212.444,Z 376.13,A -85,B 0,C 180,E1 -20782.397,E2 -20782.397} C_VEL
LIN {X 0,Y 212.07,Z 377.518,A -85,B 0,C 180,E1 -20784.295,E2 -20784.295} C_VEL
LIN {X 0,Y 211.852,Z 378.504,A -85,B 0,C 180,E1 -20786.197,E2 -20786.197} C_VEL
LIN {X 0,Y 211.661,Z 379.339,A -85,B 0,C 180,E1 -20790.001,E2 -20790.001} C_VEL
LIN {X 0,Y 211.696,Z 379.146,A -85,B 0,C 180,E1 -20791.903,E2 -20791.903} C_VEL
LIN {X 0,Y 211.848,Z 378.561,A -85,B 0,C 180,E1 -20793.805,E2 -20793.805} C_VEL
LIN {X 0,Y 212.444,Z 376.243,A -85,B 0,C 180,E1 -20797.605,E2 -20797.605} C_VEL
LIN {X 0,Y 213.22,Z 373.383,A -85,B 0,C 180,E1 -20800.446,E2 -20800.446} C_VEL
LIN {X 0,Y 214.442,Z 369.499,A -85,B 0,C 180,E1 -20803.263,E2 -20803.263} C_VEL
LIN {X 0,Y 216.108,Z 364.485,A -85,B 0,C 180,E1 -20806.048,E2 -20806.048} C_VEL
LIN {X 0,Y 218.117,Z 358.17,A -85,B 0,C 180,E1 -20808.798,E2 -20808.798} C_VEL
LIN {X 0,Y 220.67,Z 350.259,A -85,B 0,C 180,E1 -20811.486,E2 -20811.486} C_VEL
LIN {X 0,Y 223.002,Z 342.245,A -85,B 0,C 180,E1 -20813.679,E2 -20813.679} C_VEL
LIN {X 0,Y 225.51,Z 332.36,A -85,B 0,C 180,E1 -20815.869,E2 -20815.869} C_VEL
LIN {X 0,Y 228.181,Z 321.271,A -85,B 0,C 180,E1 -20817.766,E2 -20817.766} C_VEL
LIN {X 0,Y 230.349,Z 310.399,A -85,B 0,C 180,E1 -20819.221,E2 -20819.221} C_VEL
LIN {X 0,Y 232.238,Z 298.381,A -85,B 0,C 180,E1 -20820.457,E2 -20820.457} C_VEL
LIN {X 0,Y 233.722,Z 285.973,A -85,B 0,C 180,E1 -20821.374,E2 -20821.374} C_VEL
LIN {X 0,Y 234.769,Z 273.282,A -85,B 0,C 180,E1 -20821.965,E2 -20821.965} C_VEL
LIN {X 0,Y 237.079,Z 216.963,A -85,B 0,C 180,E1 -20823.626,E2 -20823.626} C_VEL
LIN {X 0,Y 231.162,Z 202.883,A -85,B 0,C 180,E1 -20825.14,E2 -20825.14} C_VEL
LIN {X 0,Y 226.238,Z 193.015,A -85,B 0,C 180,E1 -20826.412,E2 -20826.412} C_VEL
LIN {X 0,Y 218.457,Z 180.11,A -85,B 0,C 180,E1 -20828.476,E2 -20828.476} C_VEL
LIN {X 0,Y 215.892,Z 176.137,A -85,B 0,C 180,E1 -20829.191,E2 -20829.191} C_VEL
LIN {X 0,Y 214.28,Z 173.797,A -85,B 0,C 180,E1 -20829.646,E2 -20829.646} C_VEL
LIN {X 0,Y 213.728,Z 171.86,A -85,B 0,C 180,E1 -20829.902,E2 -20829.902} C_VEL
LIN {X 0,Y 213.702,Z 171.867,A -85,B 0,C 180,E1 -20833.68,E2 -20833.68} C_VEL
LIN {X 0,Y 213.702,Z 171.859,A -85,B 0,C 180,E1 -20836.346,E2 -20836.346} C_VEL
LIN {X 0,Y 213.705,Z 171.859,A -85,B 0,C 180,E1 -20841.329,E2 -20841.329} C_VEL
LIN {X 0,Y 213.755,Z 171.85,A -85,B 0,C 180,E1 -20846.017,E2 -20846.017} C_VEL
LIN {X 0,Y 213.751,Z 171.845,A -85,B 0,C 180,E1 -20850.449,E2 -20850.449} C_VEL
LIN {X 0,Y 213.783,Z 171.855,A -85,B 0,C 180,E1 -20854.699,E2 -20854.699} C_VEL
LIN {X 0,Y 213.794,Z 171.841,A -85,B 0,C 180,E1 -20858.801,E2 -20858.801} C_VEL
LIN {X 0,Y 213.882,Z 171.836,A -85,B 0,C 180,E1 -20862.798,E2 -20862.798} C_VEL
LIN {X 0,Y 213.915,Z 171.828,A -85,B 0,C 180,E1 -20866.704,E2 -20866.704} C_VEL
LIN {X 0,Y 214.134,Z 171.805,A -85,B 0,C 180,E1 -20870.555,E2 -20870.555} C_VEL
LIN {X 0,Y 214.071,Z 171.803,A -85,B 0,C 180,E1 -20874.348,E2 -20874.348} C_VEL
LIN {X 0,Y 214.403,Z 171.776,A -85,B 0,C 180,E1 -20878.121,E2 -20878.121} C_VEL
LIN {X 0,Y 214.511,Z 171.747,A -85,B 0,C 180,E1 -20880,E2 -20880} C_VEL
LIN {X 0,Y 214.4,Z 171.757,A -85,B 0,C 180,E1 -20881.878,E2 -20881.878} C_VEL
LIN {X 0,Y 214.171,Z 171.796,A -85,B 0,C 180,E1 -20887.542,E2 -20887.542} C_VEL
LIN {X 0,Y 213.977,Z 171.822,A -85,B 0,C 180,E1 -20891.365,E2 -20891.365} C_VEL
LIN {X 0,Y 213.858,Z 171.834,A -85,B 0,C 180,E1 -20895.242,E2 -20895.242} C_VEL
LIN {X 0,Y 213.788,Z 171.851,A -85,B 0,C 180,E1 -20899.192,E2 -20899.192} C_VEL
LIN {X 0,Y 213.765,Z 171.843,A -85,B 0,C 180,E1 -20903.237,E2 -20903.237} C_VEL
LIN {X 0,Y 213.786,Z 171.85,A -85,B 0,C 180,E1 -20907.426,E2 -20907.426} C_VEL
LIN {X 0,Y 213.759,Z 171.858,A -85,B 0,C 180,E1 -20911.739,E2 -20911.739} C_VEL
LIN {X 0,Y 213.742,Z 171.86,A -85,B 0,C 180,E1 -20916.289,E2 -20916.289} C_VEL
LIN {X 0,Y 213.698,Z 171.861,A -85,B 0,C 180,E1 -20921.129,E2 -20921.129} C_VEL
LIN {X 0,Y 213.665,Z 171.863,A -85,B 0,C 180,E1 -20923.091,E2 -20923.091} C_VEL
LIN {X 0,Y 213.118,Z 172.336,A -85,B 0,C 180,E1 -20924.137,E2 -20924.137} C_VEL
LIN {X 0,Y 211.303,Z 174.002,A -85,B 0,C 180,E1 -20925.43,E2 -20925.43} C_VEL
LIN {X 0,Y 208.66,Z 177.654,A -85,B 0,C 180,E1 -20927.31,E2 -20927.31} C_VEL
LIN {X 0,Y 208.491,Z 179.563,A -85,B 0,C 180,E1 -20928.297,E2 -20928.297} C_VEL
LIN {X 0,Y 208.845,Z 180.764,A -85,B 0,C 180,E1 -20928.939,E2 -20928.939} C_VEL
LIN {X 0,Y 211.267,Z 185.193,A -85,B 0,C 180,E1 -20929.697,E2 -20929.697} C_VEL
LIN {X 0,Y 217.109,Z 196.305,A -85,B 0,C 180,E1 -20931.442,E2 -20931.442} C_VEL
LIN {X 0,Y 223.716,Z 210.589,A -85,B 0,C 180,E1 -20933.328,E2 -20933.328} C_VEL
LIN {X 0,Y 227.818,Z 221.116,A -85,B 0,C 180,E1 -20934.485,E2 -20934.485} C_VEL
LIN {X 0,Y 230.215,Z 239.824,A -85,B 0,C 180,E1 -20935.6,E2 -20935.6} C_VEL
LIN {X 0,Y 228.001,Z 290.49,A -85,B 0,C 180,E1 -20937.157,E2 -20937.157} C_VEL
LIN {X 0,Y 226.579,Z 303.985,A -85,B 0,C 180,E1 -20937.88,E2 -20937.88} C_VEL
LIN {X 0,Y 224.536,Z 316.808,A -85,B 0,C 180,E1 -20938.905,E2 -20938.905} C_VEL
LIN {X 0,Y 221.985,Z 329.484,A -85,B 0,C 180,E1 -20940.35,E2 -20940.35} C_VEL
LIN {X 0,Y 219.27,Z 340.761,A -85,B 0,C 180,E1 -20942.046,E2 -20942.046} C_VEL
LIN {X 0,Y 216.506,Z 350.924,A -85,B 0,C 180,E1 -20944.009,E2 -20944.009} C_VEL
LIN {X 0,Y 213.769,Z 360.084,A -85,B 0,C 180,E1 -20946.25,E2 -20946.25} C_VEL
LIN {X 0,Y 211.02,Z 369.422,A -85,B 0,C 180,E1 -20949.169,E2 -20949.169} C_VEL
LIN {X 0,Y 208.814,Z 376.218,A -85,B 0,C 180,E1 -20951.86,E2 -20951.86} C_VEL
LIN {X 0,Y 206.681,Z 382.773,A -85,B 0,C 180,E1 -20955.224,E2 -20955.224} C_VEL
LIN {X 0,Y 205.492,Z 387.121,A -85,B 0,C 180,E1 -20958.158,E2 -20958.158} C_VEL
LIN {X 0,Y 204.965,Z 389.427,A -85,B 0,C 180,E1 -20960.127,E2 -20960.127} C_VEL
LIN {X 0,Y 204.571,Z 391.294,A -85,B 0,C 180,E1 -20962.101,E2 -20962.101} C_VEL
LIN {X 0,Y 204.353,Z 393.612,A -85,B 0,C 180,E1 -20965.833,E2 -20965.833} C_VEL
LIN {X 0,Y 204.409,Z 394.319,A -85,B 0,C 180,E1 -20968.029,E2 -20968.029} C_VEL
LIN {X 0,Y 204.534,Z 394.537,A -85,B 0,C 180,E1 -20969.999,E2 -20969.999} C_VEL
LIN {X 0,Y 204.409,Z 394.307,A -85,B 0,C 180,E1 -20971.969,E2 -20971.969} C_VEL
LIN {X 0,Y 204.346,Z 393.602,A -85,B 0,C 180,E1 -20974.143,E2 -20974.143} C_VEL
LIN {X 0,Y 204.601,Z 391.257,A -85,B 0,C 180,E1 -20977.896,E2 -20977.896} C_VEL
LIN {X 0,Y 205.207,Z 388.293,A -85,B 0,C 180,E1 -20980.856,E2 -20980.856} C_VEL
LIN {X 0,Y 206.185,Z 384.288,A -85,B 0,C 180,E1 -20983.803,E2 -20983.803} C_VEL
LIN {X 0,Y 208.18,Z 378.15,A -85,B 0,C 180,E1 -20987.18,E2 -20987.18} C_VEL
LIN {X 0,Y 210.325,Z 371.524,A -85,B 0,C 180,E1 -20989.998,E2 -20989.998} C_VEL
LIN {X 0,Y 212.785,Z 363.289,A -85,B 0,C 180,E1 -20992.783,E2 -20992.783} C_VEL
LIN {X 0,Y 215.33,Z 354.621,A -85,B 0,C 180,E1 -20995.105,E2 -20995.105} C_VEL
LIN {X 0,Y 218.304,Z 344.108,A -85,B 0,C 180,E1 -20997.305,E2 -20997.305} C_VEL
LIN {X 0,Y 221.248,Z 332.275,A -85,B 0,C 180,E1 -20999.233,E2 -20999.233} C_VEL
LIN {X 0,Y 223.802,Z 320.355,A -85,B 0,C 180,E1 -21000.682,E2 -21000.682} C_VEL
LIN {X 0,Y 225.925,Z 307.948,A -85,B 0,C 180,E1 -21001.794,E2 -21001.794} C_VEL
LIN {X 0,Y 227.519,Z 295.037,A -85,B 0,C 180,E1 -21002.597,E2 -21002.597} C_VEL
LIN {X 0,Y 228.362,Z 280.316,A -85,B 0,C 180,E1 -21003.155,E2 -21003.155} C_VEL
LIN {X 0,Y 230.066,Z 239.531,A -85,B 0,C 180,E1 -21004.375,E2 -21004.375} C_VEL
LIN {X 0,Y 227.545,Z 220.185,A -85,B 0,C 180,E1 -21005.535,E2 -21005.535} C_VEL
LIN {X 0,Y 221.204,Z 204.949,A -85,B 0,C 180,E1 -21007.309,E2 -21007.309} C_VEL
LIN {X 0,Y 213.867,Z 189.862,A -85,B 0,C 180,E1 -21009.444,E2 -21009.444} C_VEL
LIN {X 0,Y 210.64,Z 184.269,A -85,B 0,C 180,E1 -21010.406,E2 -21010.406} C_VEL
LIN {X 0,Y 208.799,Z 180.609,A -85,B 0,C 180,E1 -21011.046,E2 -21011.046} C_VEL
LIN {X 0,Y 206.651,Z 172.745,A -85,B 0,C 180,E1 -21015.574,E2 -21015.574} C_VEL
LIN {X 0,Y 206.642,Z 172.74,A -85,B 0,C 180,E1 -21019.744,E2 -21019.744} C_VEL
LIN {X 0,Y 206.695,Z 172.737,A -85,B 0,C 180,E1 -21024.688,E2 -21024.688} C_VEL
LIN {X 0,Y 206.69,Z 172.736,A -85,B 0,C 180,E1 -21029.333,E2 -21029.333} C_VEL
LIN {X 0,Y 206.68,Z 172.737,A -85,B 0,C 180,E1 -21033.765,E2 -21033.765} C_VEL
LIN {X 0,Y 206.706,Z 172.725,A -85,B 0,C 180,E1 -21038.038,E2 -21038.038} C_VEL
LIN {X 0,Y 206.797,Z 172.715,A -85,B 0,C 180,E1 -21042.19,E2 -21042.19} C_VEL
LIN {X 0,Y 206.844,Z 172.719,A -85,B 0,C 180,E1 -21046.241,E2 -21046.241} C_VEL
LIN {X 0,Y 207.065,Z 172.675,A -85,B 0,C 180,E1 -21050.229,E2 -21050.229} C_VEL
LIN {X 0,Y 207.023,Z 172.698,A -85,B 0,C 180,E1 -21054.155,E2 -21054.155} C_VEL
LIN {X 0,Y 207.332,Z 172.641,A -85,B 0,C 180,E1 -21058.058,E2 -21058.058} C_VEL
LIN {X 0,Y 207.472,Z 172.638,A -85,B 0,C 180,E1 -21060,E2 -21060} C_VEL
LIN {X 0,Y 207.336,Z 172.657,A -85,B 0,C 180,E1 -21061.943,E2 -21061.943} C_VEL
LIN {X 0,Y 207.12,Z 172.683,A -85,B 0,C 180,E1 -21067.801,E2 -21067.801} C_VEL
LIN {X 0,Y 206.891,Z 172.696,A -85,B 0,C 180,E1 -21071.76,E2 -21071.76} C_VEL
LIN {X 0,Y 206.798,Z 172.727,A -85,B 0,C 180,E1 -21075.776,E2 -21075.776} C_VEL
LIN {X 0,Y 206.706,Z 172.721,A -85,B 0,C 180,E1 -21079.877,E2 -21079.877} C_VEL
LIN {X 0,Y 206.722,Z 172.731,A -85,B 0,C 180,E1 -21084.077,E2 -21084.077} C_VEL
LIN {X 0,Y 206.682,Z 172.739,A -85,B 0,C 180,E1 -21088.428,E2 -21088.428} C_VEL
LIN {X 0,Y 206.689,Z 172.732,A -85,B 0,C 180,E1 -21092.96,E2 -21092.96} C_VEL
LIN {X 0,Y 206.663,Z 172.739,A -85,B 0,C 180,E1 -21097.744,E2 -21097.744} C_VEL
LIN {X 0,Y 206.628,Z 172.745,A -85,B 0,C 180,E1 -21101.561,E2 -21101.561} C_VEL
LIN {X 0,Y 206.627,Z 172.739,A -85,B 0,C 180,E1 -21105.584,E2 -21105.584} C_VEL
LIN {X 0,Y 206.645,Z 172.738,A -85,B 0,C 180,E1 -21108.654,E2 -21108.654} C_VEL
LIN {X 0,Y 207.761,Z 175.743,A -85,B 0,C 180,E1 -21109.098,E2 -21109.098} C_VEL
LIN {X 0,Y 209.59,Z 178.029,A -85,B 0,C 180,E1 -21109.635,E2 -21109.635} C_VEL
LIN {X 0,Y 216.99,Z 189.718,A -85,B 0,C 180,E1 -21111.778,E2 -21111.778} C_VEL
LIN {X 0,Y 223.41,Z 201.186,A -85,B 0,C 180,E1 -21113.528,E2 -21113.528} C_VEL
LIN {X 0,Y 229.076,Z 213.885,A -85,B 0,C 180,E1 -21115.058,E2 -21115.058} C_VEL
LIN {X 0,Y 231.031,Z 218.744,A -85,B 0,C 180,E1 -21115.58,E2 -21115.58} C_VEL
LIN {X 0,Y 228.437,Z 276.802,A -85,B 0,C 180,E1 -21117.352,E2 -21117.352} C_VEL
LIN {X 0,Y 227.239,Z 289.684,A -85,B 0,C 180,E1 -21118.068,E2 -21118.068} C_VEL
LIN {X 0,Y 225.538,Z 301.848,A -85,B 0,C 180,E1 -21119.061,E2 -21119.061} C_VEL
LIN {X 0,Y 223.594,Z 313.14,A -85,B 0,C 180,E1 -21120.328,E2 -21120.328} C_VEL
LIN {X 0,Y 220.99,Z 324.764,A -85,B 0,C 180,E1 -21122.027,E2 -21122.027} C_VEL
LIN {X 0,Y 218.602,Z 334.346,A -85,B 0,C 180,E1 -21123.817,E2 -21123.817} C_VEL
LIN {X 0,Y 216.114,Z 343.881,A -85,B 0,C 180,E1 -21126.065,E2 -21126.065} C_VEL
LIN {X 0,Y 213.697,Z 351.567,A -85,B 0,C 180,E1 -21128.287,E2 -21128.287} C_VEL
LIN {X 0,Y 211.087,Z 359.239,A -85,B 0,C 180,E1 -21131.059,E2 -21131.059} C_VEL
LIN {X 0,Y 208.699,Z 366.278,A -85,B 0,C 180,E1 -21134.373,E2 -21134.373} C_VEL
LIN {X 0,Y 207.1,Z 370.962,A -85,B 0,C 180,E1 -21137.258,E2 -21137.258} C_VEL
LIN {X 0,Y 205.92,Z 374.543,A -85,B 0,C 180,E1 -21140.176,E2 -21140.176} C_VEL
LIN {X 0,Y 205.069,Z 377.513,A -85,B 0,C 180,E1 -21143.656,E2 -21143.656} C_VEL
LIN {X 0,Y 204.766,Z 378.764,A -85,B 0,C 180,E1 -21146.065,E2 -21146.065} C_VEL
LIN {X 0,Y 204.618,Z 379.37,A -85,B 0,C 180,E1 -21148.033,E2 -21148.033} C_VEL
LIN {X 0,Y 204.578,Z 379.598,A -85,B 0,C 180,E1 -21150.001,E2 -21150.001} C_VEL
LIN {X 0,Y 204.617,Z 379.404,A -85,B 0,C 180,E1 -21151.969,E2 -21151.969} C_VEL
LIN {X 0,Y 204.763,Z 378.82,A -85,B 0,C 180,E1 -21153.937,E2 -21153.937} C_VEL
LIN {X 0,Y 205.411,Z 376.501,A -85,B 0,C 180,E1 -21157.867,E2 -21157.867} C_VEL
LIN {X 0,Y 206.243,Z 373.641,A -85,B 0,C 180,E1 -21160.803,E2 -21160.803} C_VEL
LIN {X 0,Y 207.547,Z 369.757,A -85,B 0,C 180,E1 -21163.712,E2 -21163.712} C_VEL
LIN {X 0,Y 209.294,Z 364.743,A -85,B 0,C 180,E1 -21166.585,E2 -21166.585} C_VEL
LIN {X 0,Y 211.41,Z 358.427,A -85,B 0,C 180,E1 -21169.417,E2 -21169.417} C_VEL
LIN {X 0,Y 214.089,Z 350.516,A -85,B 0,C 180,E1 -21172.181,E2 -21172.181} C_VEL
LIN {X 0,Y 216.638,Z 342.084,A -85,B 0,C 180,E1 -21174.54,E2 -21174.54} C_VEL
LIN {X 0,Y 219.157,Z 332.615,A -85,B 0,C 180,E1 -21176.677,E2 -21176.677} C_VEL
LIN {X 0,Y 221.631,Z 322.918,A -85,B 0,C 180,E1 -21178.403,E2 -21178.403} C_VEL
LIN {X 0,Y 223.88,Z 312.412,A -85,B 0,C 180,E1 -21179.891,E2 -21179.891} C_VEL
LIN {X 0,Y 225.966,Z 299.76,A -85,B 0,C 180,E1 -21181.267,E2 -21181.267} C_VEL
LIN {X 0,Y 227.599,Z 287.21,A -85,B 0,C 180,E1 -21182.239,E2 -21182.239} C_VEL
LIN {X 0,Y 228.736,Z 274.642,A -85,B 0,C 180,E1 -21182.864,E2 -21182.864} C_VEL
LIN {X 0,Y 231.173,Z 218.945,A -85,B 0,C 180,E1 -21184.541,E2 -21184.541} C_VEL
LIN {X 0,Y 225.011,Z 204.422,A -85,B 0,C 180,E1 -21186.2,E2 -21186.2} C_VEL
LIN {X 0,Y 220.125,Z 194.931,A -85,B 0,C 180,E1 -21187.527,E2 -21187.527} C_VEL
LIN {X 0,Y 213.365,Z 184.004,A -85,B 0,C 180,E1 -21189.413,E2 -21189.413} C_VEL
LIN {X 0,Y 211.062,Z 180.464,A -85,B 0,C 180,E1 -21190.088,E2 -21190.088} C_VEL
LIN {X 0,Y 209.02,Z 177.172,A -85,B 0,C 180,E1 -21190.711,E2 -21190.711} C_VEL
LIN {X 0,Y 207.241,Z 174.811,A -85,B 0,C 180,E1 -21191.246,E2 -21191.246} C_VEL
LIN {X 0,Y 206.631,Z 172.746,A -85,B 0,C 180,E1 -21191.541,E2 -21191.541} C_VEL
LIN {X 0,Y 206.631,Z 172.737,A -85,B 0,C 180,E1 -21195.583,E2 -21195.583} C_VEL
LIN {X 0,Y 206.648,Z 172.732,A -85,B 0,C 180,E1 -21199.745,E2 -21199.745} C_VEL
LIN {X 0,Y 206.701,Z 172.724,A -85,B 0,C 180,E1 -21204.689,E2 -21204.689} C_VEL
LIN {X 0,Y 206.697,Z 172.73,A -85,B 0,C 180,E1 -21209.334,E2 -21209.334} C_VEL
LIN {X 0,Y 206.707,Z 172.736,A -85,B 0,C 180,E1 -21213.768,E2 -21213.768} C_VEL
LIN {X 0,Y 206.731,Z 172.715,A -85,B 0,C 180,E1 -21218.04,E2 -21218.04} C_VEL
LIN {X 0,Y 206.823,Z 172.72,A -85,B 0,C 180,E1 -21222.192,E2 -21222.192} C_VEL
LIN {X 0,Y 206.855,Z 172.703,A -85,B 0,C 180,E1 -21226.241,E2 -21226.241} C_VEL
LIN {X 0,Y 207.079,Z 172.686,A -85,B 0,C 180,E1 -21230.23,E2 -21230.23} C_VEL
LIN {X 0,Y 207.035,Z 172.677,A -85,B 0,C 180,E1 -21234.155,E2 -21234.155} C_VEL
LIN {X 0,Y 207.343,Z 172.656,A -85,B 0,C 180,E1 -21238.057,E2 -21238.057} C_VEL
LIN {X 0,Y 207.479,Z 172.622,A -85,B 0,C 180,E1 -21240,E2 -21240} C_VEL
LIN {X 0,Y 207.339,Z 172.635,A -85,B 0,C 180,E1 -21241.942,E2 -21241.942} C_VEL
LIN {X 0,Y 207.116,Z 172.671,A -85,B 0,C 180,E1 -21247.801,E2 -21247.801} C_VEL
LIN {X 0,Y 206.896,Z 172.706,A -85,B 0,C 180,E1 -21251.76,E2 -21251.76} C_VEL
LIN {X 0,Y 206.792,Z 172.708,A -85,B 0,C 180,E1 -21255.777,E2 -21255.777} C_VEL
LIN {X 0,Y 206.71,Z 172.736,A -85,B 0,C 180,E1 -21259.876,E2 -21259.876} C_VEL
LIN {X 0,Y 206.692,Z 172.726,A -85,B 0,C 180,E1 -21264.081,E2 -21264.081} C_VEL
LIN {X 0,Y 206.687,Z 172.728,A -85,B 0,C 180,E1 -21268.427,E2 -21268.427} C_VEL
LIN {X 0,Y 206.695,Z 172.731,A -85,B 0,C 180,E1 -21272.958,E2 -21272.958} C_VEL
LIN {X 0,Y 206.667,Z 172.733,A -85,B 0,C 180,E1 -21277.743,E2 -21277.743} C_VEL
LIN {X 0,Y 206.632,Z 172.74,A -85,B 0,C 180,E1 -21281.559,E2 -21281.559} C_VEL
LIN {X 0,Y 206.661,Z 172.775,A -85,B 0,C 180,E1 -21284.426,E2 -21284.426} C_VEL
LIN {X 0,Y 208.491,Z 179.563,A -85,B 0,C 180,E1 -21288.297,E2 -21288.297} C_VEL
LIN {X 0,Y 209.301,Z 181.516,A -85,B 0,C 180,E1 -21288.975,E2 -21288.975} C_VEL
LIN {X 0,Y 211.026,Z 185.791,A -85,B 0,C 180,E1 -21289.668,E2 -21289.668} C_VEL
LIN {X 0,Y 212.448,Z 192.215,A -85,B 0,C 180,E1 -21290.266,E2 -21290.266} C_VEL
LIN {X 0,Y 213.721,Z 200.305,A -85,B 0,C 180,E1 -21290.845,E2 -21290.845} C_VEL
LIN {X 0,Y 215.06,Z 206.06,A -85,B 0,C 180,E1 -21291.412,E2 -21291.412} C_VEL
LIN {X 0,Y 215.778,Z 207.825,A -85,B 0,C 180,E1 -21291.641,E2 -21291.641} C_VEL
LIN {X 0,Y 221.663,Z 221.898,A -85,B 0,C 180,E1 -21293.382,E2 -21293.382} C_VEL
LIN {X 0,Y 222.339,Z 224.765,A -85,B 0,C 180,E1 -21293.623,E2 -21293.623} C_VEL
LIN {X 0,Y 224.335,Z 241.228,A -85,B 0,C 180,E1 -21294.628,E2 -21294.628} C_VEL
LIN {X 0,Y 222.09,Z 289.829,A -85,B 0,C 180,E1 -21296.142,E2 -21296.142} C_VEL
LIN {X 0,Y 220.683,Z 303.157,A -85,B 0,C 180,E1 -21296.862,E2 -21296.862} C_VEL
LIN {X 0,Y 218.699,Z 315.449,A -85,B 0,C 180,E1 -21297.842,E2 -21297.842} C_VEL
LIN {X 0,Y 216.199,Z 327.645,A -85,B 0,C 180,E1 -21299.203,E2 -21299.203} C_VEL
LIN {X 0,Y 213.373,Z 339.211,A -85,B 0,C 180,E1 -21300.933,E2 -21300.933} C_VEL
LIN {X 0,Y 210.419,Z 349.63,A -85,B 0,C 180,E1 -21302.93,E2 -21302.93} C_VEL
LIN {X 0,Y 207.791,Z 358.154,A -85,B 0,C 180,E1 -21304.989,E2 -21304.989} C_VEL
LIN {X 0,Y 205.338,Z 366.026,A -85,B 0,C 180,E1 -21307.352,E2 -21307.352} C_VEL
LIN {X 0,Y 202.802,Z 373.719,A -85,B 0,C 180,E1 -21310.251,E2 -21310.251} C_VEL
LIN {X 0,Y 201.03,Z 378.995,A -85,B 0,C 180,E1 -21312.712,E2 -21312.712} C_VEL
LIN {X 0,Y 199.259,Z 384.107,A -85,B 0,C 180,E1 -21315.705,E2 -21315.705} C_VEL
LIN {X 0,Y 198.198,Z 388.089,A -85,B 0,C 180,E1 -21318.753,E2 -21318.753} C_VEL
LIN {X 0,Y 197.511,Z 391.034,A -85,B 0,C 180,E1 -21321.816,E2 -21321.816} C_VEL
LIN {X 0,Y 197.306,Z 392.439,A -85,B 0,C 180,E1 -21323.865,E2 -21323.865} C_VEL
LIN {X 0,Y 197.252,Z 393.502,A -85,B 0,C 180,E1 -21326.056,E2 -21326.056} C_VEL
LIN {X 0,Y 197.451,Z 394.278,A -85,B 0,C 180,E1 -21329.999,E2 -21329.999} C_VEL
LIN {X 0,Y 197.248,Z 393.487,A -85,B 0,C 180,E1 -21333.928,E2 -21333.928} C_VEL
LIN {X 0,Y 197.332,Z 392.412,A -85,B 0,C 180,E1 -21336.132,E2 -21336.132} C_VEL
LIN {X 0,Y 197.535,Z 390.995,A -85,B 0,C 180,E1 -21338.181,E2 -21338.181} C_VEL
LIN {X 0,Y 198.201,Z 388.031,A -85,B 0,C 180,E1 -21341.245,E2 -21341.245} C_VEL
LIN {X 0,Y 199.257,Z 384.027,A -85,B 0,C 180,E1 -21344.293,E2 -21344.293} C_VEL
LIN {X 0,Y 201.382,Z 377.888,A -85,B 0,C 180,E1 -21347.779,E2 -21347.779} C_VEL
LIN {X 0,Y 203.835,Z 370.699,A -85,B 0,C 180,E1 -21350.903,E2 -21350.903} C_VEL
LIN {X 0,Y 206.251,Z 362.876,A -85,B 0,C 180,E1 -21353.601,E2 -21353.601} C_VEL
LIN {X 0,Y 208.914,Z 354.359,A -85,B 0,C 180,E1 -21355.932,E2 -21355.932} C_VEL
LIN {X 0,Y 212.005,Z 343.844,A -85,B 0,C 180,E1 -21358.188,E2 -21358.188} C_VEL
LIN {X 0,Y 215.074,Z 332.011,A -85,B 0,C 180,E1 -21360.158,E2 -21360.158} C_VEL
LIN {X 0,Y 217.733,Z 320.09,A -85,B 0,C 180,E1 -21361.634,E2 -21361.634} C_VEL
LIN {X 0,Y 219.915,Z 307.68,A -85,B 0,C 180,E1 -21362.769,E2 -21362.769} C_VEL
LIN {X 0,Y 221.526,Z 295.142,A -85,B 0,C 180,E1 -21363.567,E2 -21363.567} C_VEL
LIN {X 0,Y 222.39,Z 281.232,A -85,B 0,C 180,E1 -21364.121,E2 -21364.121} C_VEL
LIN {X 0,Y 224.214,Z 240.964,A -85,B 0,C 180,E1 -21365.338,E2 -21365.338} C_VEL
LIN {X 0,Y 221.923,Z 222.678,A -85,B 0,C 180,E1 -21366.469,E2 -21366.469} C_VEL
LIN {X 0,Y 215.437,Z 207.09,A -85,B 0,C 180,E1 -21368.386,E2 -21368.386} C_VEL
LIN {X 0,Y 208.822,Z 193.626,A -85,B 0,C 180,E1 -21370.414,E2 -21370.414} C_VEL
LIN {X 0,Y 203.75,Z 184.609,A -85,B 0,C 180,E1 -21372.044,E2 -21372.044} C_VEL
LIN {X 0,Y 201.419,Z 180.281,A -85,B 0,C 180,E1 -21372.883,E2 -21372.883} C_VEL
LIN {X 0,Y 199.571,Z 173.622,A -85,B 0,C 180,E1 -21376.966,E2 -21376.966} C_VEL
LIN {X 0,Y 199.592,Z 173.622,A -85,B 0,C 180,E1 -21380.772,E2 -21380.772} C_VEL
LIN {X 0,Y 199.605,Z 173.617,A -85,B 0,C 180,E1 -21385.712,E2 -21385.712} C_VEL
LIN {X 0,Y 199.68,Z 173.605,A -85,B 0,C 180,E1 -21388.133,E2 -21388.133} C_VEL
LIN {X 0,Y 199.629,Z 173.606,A -85,B 0,C 180,E1 -21392.763,E2 -21392.763} C_VEL
LIN {X 0,Y 199.664,Z 173.598,A -85,B 0,C 180,E1 -21397.22,E2 -21397.22} C_VEL
LIN {X 0,Y 199.739,Z 173.597,A -85,B 0,C 180,E1 -21401.802,E2 -21401.802} C_VEL
LIN {X 0,Y 199.762,Z 173.599,A -85,B 0,C 180,E1 -21405.743,E2 -21405.743} C_VEL
LIN {X 0,Y 200.017,Z 173.553,A -85,B 0,C 180,E1 -21409.882,E2 -21409.882} C_VEL
LIN {X 0,Y 199.987,Z 173.575,A -85,B 0,C 180,E1 -21413.948,E2 -21413.948} C_VEL
LIN {X 0,Y 200.274,Z 173.519,A -85,B 0,C 180,E1 -21417.989,E2 -21417.989} C_VEL
LIN {X 0,Y 200.439,Z 173.514,A -85,B 0,C 180,E1 -21420,E2 -21420} C_VEL
LIN {X 0,Y 199.979,Z 173.557,A -85,B 0,C 180,E1 -21424.031,E2 -21424.031} C_VEL
LIN {X 0,Y 200.068,Z 173.564,A -85,B 0,C 180,E1 -21428.078,E2 -21428.078} C_VEL
LIN {X 0,Y 199.999,Z 173.567,A -85,B 0,C 180,E1 -21430.298,E2 -21430.298} C_VEL
LIN {X 0,Y 199.737,Z 173.604,A -85,B 0,C 180,E1 -21436.349,E2 -21436.349} C_VEL
LIN {X 0,Y 199.639,Z 173.605,A -85,B 0,C 180,E1 -21440.612,E2 -21440.612} C_VEL
LIN {X 0,Y 199.636,Z 173.606,A -85,B 0,C 180,E1 -21444.99,E2 -21444.99} C_VEL
LIN {X 0,Y 199.603,Z 173.62,A -85,B 0,C 180,E1 -21449.534,E2 -21449.534} C_VEL
LIN {X 0,Y 199.66,Z 173.604,A -85,B 0,C 180,E1 -21452.353,E2 -21452.353} C_VEL
LIN {X 0,Y 199.612,Z 173.622,A -85,B 0,C 180,E1 -21456.766,E2 -21456.766} C_VEL
LIN {X 0,Y 199.59,Z 173.622,A -85,B 0,C 180,E1 -21459.333,E2 -21459.333} C_VEL
LIN {X 0,Y 199.563,Z 173.624,A -85,B 0,C 180,E1 -21462.309,E2 -21462.309} C_VEL
LIN {X 0,Y 199.573,Z 173.626,A -85,B 0,C 180,E1 -21466.857,E2 -21466.857} C_VEL
LIN {X 0,Y 200.549,Z 176.437,A -85,B 0,C 180,E1 -21467.302,E2 -21467.302} C_VEL
LIN {X 0,Y 202.724,Z 179.148,A -85,B 0,C 180,E1 -21468,E2 -21468} C_VEL
LIN {X 0,Y 210.749,Z 191.549,A -85,B 0,C 180,E1 -21470.495,E2 -21470.495} C_VEL
LIN {X 0,Y 217.848,Z 203.837,A -85,B 0,C 180,E1 -21472.536,E2 -21472.536} C_VEL
LIN {X 0,Y 223.835,Z 217.369,A -85,B 0,C 180,E1 -21474.241,E2 -21474.241} C_VEL
LIN {X 0,Y 225.118,Z 220.649,A -85,B 0,C 180,E1 -21474.604,E2 -21474.604} C_VEL
LIN {X 0,Y 222.511,Z 276.924,A -85,B 0,C 180,E1 -21476.36,E2 -21476.36} C_VEL
LIN {X 0,Y 221.227,Z 290.048,A -85,B 0,C 180,E1 -21477.101,E2 -21477.101} C_VEL
LIN {X 0,Y 219.496,Z 302.114,A -85,B 0,C 180,E1 -21478.11,E2 -21478.11} C_VEL
LIN {X 0,Y 217.474,Z 313.404,A -85,B 0,C 180,E1 -21479.405,E2 -21479.405} C_VEL
LIN {X 0,Y 214.768,Z 325.026,A -85,B 0,C 180,E1 -21481.141,E2 -21481.141} C_VEL
LIN {X 0,Y 211.975,Z 335.778,A -85,B 0,C 180,E1 -21483.226,E2 -21483.226} C_VEL
LIN {X 0,Y 209.579,Z 344.34,A -85,B 0,C 180,E1 -21485.328,E2 -21485.328} C_VEL
LIN {X 0,Y 206.626,Z 353.212,A -85,B 0,C 180,E1 -21488.03,E2 -21488.03} C_VEL
LIN {X 0,Y 203.997,Z 360.608,A -85,B 0,C 180,E1 -21490.897,E2 -21490.897} C_VEL
LIN {X 0,Y 201.865,Z 366.539,A -85,B 0,C 180,E1 -21493.829,E2 -21493.829} C_VEL
LIN {X 0,Y 200.192,Z 371.222,A -85,B 0,C 180,E1 -21496.811,E2 -21496.811} C_VEL
LIN {X 0,Y 198.917,Z 374.804,A -85,B 0,C 180,E1 -21499.826,E2 -21499.826} C_VEL
LIN {X 0,Y 198.376,Z 376.65,A -85,B 0,C 180,E1 -21501.854,E2 -21501.854} C_VEL
LIN {X 0,Y 197.951,Z 378.037,A -85,B 0,C 180,E1 -21503.887,E2 -21503.887} C_VEL
LIN {X 0,Y 197.541,Z 379.629,A -85,B 0,C 180,E1 -21507.962,E2 -21507.962} C_VEL
LIN {X 0,Y 197.496,Z 379.856,A -85,B 0,C 180,E1 -21510.001,E2 -21510.001} C_VEL
LIN {X 0,Y 197.54,Z 379.663,A -85,B 0,C 180,E1 -21512.04,E2 -21512.04} C_VEL
LIN {X 0,Y 197.951,Z 378.114,A -85,B 0,C 180,E1 -21516.115,E2 -21516.115} C_VEL
LIN {X 0,Y 198.376,Z 376.76,A -85,B 0,C 180,E1 -21518.148,E2 -21518.148} C_VEL
LIN {X 0,Y 199.258,Z 373.9,A -85,B 0,C 180,E1 -21521.187,E2 -21521.187} C_VEL
LIN {X 0,Y 200.668,Z 370.015,A -85,B 0,C 180,E1 -21524.192,E2 -21524.192} C_VEL
LIN {X 0,Y 202.502,Z 365,A -85,B 0,C 180,E1 -21527.158,E2 -21527.158} C_VEL
LIN {X 0,Y 204.73,Z 358.684,A -85,B 0,C 180,E1 -21530.078,E2 -21530.078} C_VEL
LIN {X 0,Y 207.543,Z 350.772,A -85,B 0,C 180,E1 -21532.919,E2 -21532.919} C_VEL
LIN {X 0,Y 210.188,Z 342.341,A -85,B 0,C 180,E1 -21535.345,E2 -21535.345} C_VEL
LIN {X 0,Y 212.834,Z 332.871,A -85,B 0,C 180,E1 -21537.536,E2 -21537.536} C_VEL
LIN {X 0,Y 215.719,Z 321.78,A -85,B 0,C 180,E1 -21539.523,E2 -21539.523} C_VEL
LIN {X 0,Y 218.088,Z 310.905,A -85,B 0,C 180,E1 -21541.039,E2 -21541.039} C_VEL
LIN {X 0,Y 220.161,Z 298.883,A -85,B 0,C 180,E1 -21542.324,E2 -21542.324} C_VEL
LIN {X 0,Y 221.774,Z 286.333,A -85,B 0,C 180,E1 -21543.286,E2 -21543.286} C_VEL
LIN {X 0,Y 222.892,Z 273.5,A -85,B 0,C 180,E1 -21543.902,E2 -21543.902} C_VEL
LIN {X 0,Y 225.298,Z 220.874,A -85,B 0,C 180,E1 -21545.51,E2 -21545.51} C_VEL
LIN {X 0,Y 219.611,Z 207.485,A -85,B 0,C 180,E1 -21547.123,E2 -21547.123} C_VEL
LIN {X 0,Y 215.03,Z 198.703,A -85,B 0,C 180,E1 -21548.428,E2 -21548.428} C_VEL
LIN {X 0,Y 208.476,Z 187.949,A -85,B 0,C 180,E1 -21550.36,E2 -21550.36} C_VEL
LIN {X 0,Y 204.375,Z 181.739,A -85,B 0,C 180,E1 -21551.639,E2 -21551.639} C_VEL
LIN {X 0,Y 201.98,Z 178.128,A -85,B 0,C 180,E1 -21552.422,E2 -21552.422} C_VEL
LIN {X 0,Y 200.202,Z 175.79,A -85,B 0,C 180,E1 -21553.005,E2 -21553.005} C_VEL
LIN {X 0,Y 199.572,Z 173.625,A -85,B 0,C 180,E1 -21553.309,E2 -21553.309} C_VEL
LIN {X 0,Y 199.571,Z 173.624,A -85,B 0,C 180,E1 -21558.003,E2 -21558.003} C_VEL
LIN {X 0,Y 199.598,Z 173.611,A -85,B 0,C 180,E1 -21560.773,E2 -21560.773} C_VEL
LIN {X 0,Y 199.611,Z 173.608,A -85,B 0,C 180,E1 -21565.713,E2 -21565.713} C_VEL
LIN {X 0,Y 199.687,Z 173.611,A -85,B 0,C 180,E1 -21568.134,E2 -21568.134} C_VEL
LIN {X 0,Y 199.644,Z 173.611,A -85,B 0,C 180,E1 -21572.765,E2 -21572.765} C_VEL
LIN {X 0,Y 199.688,Z 173.591,A -85,B 0,C 180,E1 -21577.223,E2 -21577.223} C_VEL
LIN {X 0,Y 199.747,Z 173.603,A -85,B 0,C 180,E1 -21581.802,E2 -21581.802} C_VEL
LIN {X 0,Y 199.772,Z 173.58,A -85,B 0,C 180,E1 -21585.743,E2 -21585.743} C_VEL
LIN {X 0,Y 200.024,Z 173.568,A -85,B 0,C 180,E1 -21589.882,E2 -21589.882} C_VEL
LIN {X 0,Y 199.999,Z 173.551,A -85,B 0,C 180,E1 -21593.948,E2 -21593.948} C_VEL
LIN {X 0,Y 200.285,Z 173.535,A -85,B 0,C 180,E1 -21597.989,E2 -21597.989} C_VEL
LIN {X 0,Y 200.446,Z 173.497,A -85,B 0,C 180,E1 -21600,E2 -21600} C_VEL
LIN {X 0,Y 199.98,Z 173.569,A -85,B 0,C 180,E1 -21604.03,E2 -21604.03} C_VEL
LIN {X 0,Y 200.065,Z 173.547,A -85,B 0,C 180,E1 -21608.078,E2 -21608.078} C_VEL
LIN {X 0,Y 200.006,Z 173.551,A -85,B 0,C 180,E1 -21610.297,E2 -21610.297} C_VEL
LIN {X 0,Y 199.735,Z 173.584,A -85,B 0,C 180,E1 -21616.349,E2 -21616.349} C_VEL
LIN {X 0,Y 199.641,Z 173.616,A -85,B 0,C 180,E1 -21620.612,E2 -21620.612} C_VEL
LIN {X 0,Y 199.622,Z 173.614,A -85,B 0,C 180,E1 -21624.991,E2 -21624.991} C_VEL
LIN {X 0,Y 199.608,Z 173.609,A -85,B 0,C 180,E1 -21629.533,E2 -21629.533} C_VEL
LIN {X 0,Y 199.666,Z 173.611,A -85,B 0,C 180,E1 -21632.352,E2 -21632.352} C_VEL
LIN {X 0,Y 199.617,Z 173.617,A -85,B 0,C 180,E1 -21636.764,E2 -21636.764} C_VEL
LIN {X 0,Y 199.595,Z 173.62,A -85,B 0,C 180,E1 -21639.331,E2 -21639.331} C_VEL
LIN {X 0,Y 199.631,Z 173.798,A -85,B 0,C 180,E1 -21643.1,E2 -21643.1} C_VEL
LIN {X 0,Y 201.495,Z 180.475,A -85,B 0,C 180,E1 -21647.094,E2 -21647.094} C_VEL
LIN {X 0,Y 203.913,Z 184.846,A -85,B 0,C 180,E1 -21647.92,E2 -21647.92} C_VEL
LIN {X 0,Y 209.554,Z 194.934,A -85,B 0,C 180,E1 -21649.73,E2 -21649.73} C_VEL
LIN {X 0,Y 215.425,Z 207.014,A -85,B 0,C 180,E1 -21651.534,E2 -21651.534} C_VEL
LIN {X 0,Y 215.778,Z 207.825,A -85,B 0,C 180,E1 -21651.641,E2 -21651.641} C_VEL
LIN {X 0,Y 217.018,Z 211.247,A -85,B 0,C 180,E1 -21652.038,E2 -21652.038} C_VEL
LIN {X 0,Y 217.983,Z 216.879,A -85,B 0,C 180,E1 -21652.463,E2 -21652.463} C_VEL
LIN {X 0,Y 218.207,Z 222.761,A -85,B 0,C 180,E1 -21652.745,E2 -21652.745} C_VEL
LIN {X 0,Y 218.029,Z 230.891,A -85,B 0,C 180,E1 -21653.038,E2 -21653.038} C_VEL
LIN {X 0,Y 218.235,Z 238.954,A -85,B 0,C 180,E1 -21653.402,E2 -21653.402} C_VEL
LIN {X 0,Y 218.454,Z 243.909,A -85,B 0,C 180,E1 -21653.642,E2 -21653.642} C_VEL
LIN {X 0,Y 216.164,Z 290.313,A -85,B 0,C 180,E1 -21655.127,E2 -21655.127} C_VEL
LIN {X 0,Y 214.67,Z 303.69,A -85,B 0,C 180,E1 -21655.88,E2 -21655.88} C_VEL
LIN {X 0,Y 212.527,Z 316.303,A -85,B 0,C 180,E1 -21656.931,E2 -21656.931} C_VEL
LIN {X 0,Y 209.75,Z 328.975,A -85,B 0,C 180,E1 -21658.429,E2 -21658.429} C_VEL
LIN {X 0,Y 206.84,Z 340.251,A -85,B 0,C 180,E1 -21660.202,E2 -21660.202} C_VEL
LIN {X 0,Y 203.775,Z 350.409,A -85,B 0,C 180,E1 -21662.25,E2 -21662.25} C_VEL
LIN {X 0,Y 200.783,Z 359.567,A -85,B 0,C 180,E1 -21664.609,E2 -21664.609} C_VEL
LIN {X 0,Y 198.049,Z 367.867,A -85,B 0,C 180,E1 -21667.316,E2 -21667.316} C_VEL
LIN {X 0,Y 195.676,Z 374.583,A -85,B 0,C 180,E1 -21670.049,E2 -21670.049} C_VEL
LIN {X 0,Y 193.531,Z 380.559,A -85,B 0,C 180,E1 -21673.11,E2 -21673.11} C_VEL
LIN {X 0,Y 191.926,Z 385.287,A -85,B 0,C 180,E1 -21676.229,E2 -21676.229} C_VEL
LIN {X 0,Y 190.942,Z 388.908,A -85,B 0,C 180,E1 -21679.394,E2 -21679.394} C_VEL
LIN {X 0,Y 190.473,Z 390.775,A -85,B 0,C 180,E1 -21681.512,E2 -21681.512} C_VEL
LIN {X 0,Y 190.163,Z 393.185,A -85,B 0,C 180,E1 -21685.76,E2 -21685.76} C_VEL
LIN {X 0,Y 190.214,Z 393.801,A -85,B 0,C 180,E1 -21687.881,E2 -21687.881} C_VEL
LIN {X 0,Y 190.368,Z 394.019,A -85,B 0,C 180,E1 -21689.999,E2 -21689.999} C_VEL
LIN {X 0,Y 190.169,Z 393.343,A -85,B 0,C 180,E1 -21693.775,E2 -21693.775} C_VEL
LIN {X 0,Y 190.244,Z 392.152,A -85,B 0,C 180,E1 -21696.362,E2 -21696.362} C_VEL
LIN {X 0,Y 190.492,Z 390.735,A -85,B 0,C 180,E1 -21698.485,E2 -21698.485} C_VEL
LIN {X 0,Y 191.216,Z 387.77,A -85,B 0,C 180,E1 -21701.661,E2 -21701.661} C_VEL
LIN {X 0,Y 192.346,Z 383.765,A -85,B 0,C 180,E1 -21704.818,E2 -21704.818} C_VEL
LIN {X 0,Y 194.595,Z 377.626,A -85,B 0,C 180,E1 -21708.421,E2 -21708.421} C_VEL
LIN {X 0,Y 197.085,Z 370.717,A -85,B 0,C 180,E1 -21711.53,E2 -21711.53} C_VEL
LIN {X 0,Y 199.713,Z 362.612,A -85,B 0,C 180,E1 -21714.423,E2 -21714.423} C_VEL
LIN {X 0,Y 202.52,Z 354.095,A -85,B 0,C 180,E1 -21716.815,E2 -21716.815} C_VEL
LIN {X 0,Y 205.771,Z 343.581,A -85,B 0,C 180,E1 -21719.122,E2 -21719.122} C_VEL
LIN {X 0,Y 208.949,Z 331.746,A -85,B 0,C 180,E1 -21721.139,E2 -21721.139} C_VEL
LIN {X 0,Y 211.718,Z 319.824,A -85,B 0,C 180,E1 -21722.643,E2 -21722.643} C_VEL
LIN {X 0,Y 213.976,Z 307.413,A -85,B 0,C 180,E1 -21723.799,E2 -21723.799} C_VEL
LIN {X 0,Y 215.694,Z 294.553,A -85,B 0,C 180,E1 -21724.625,E2 -21724.625} C_VEL
LIN {X 0,Y 216.632,Z 279.566,A -85,B 0,C 180,E1 -21725.214,E2 -21725.214} C_VEL
LIN {X 0,Y 218.359,Z 240.944,A -85,B 0,C 180,E1 -21726.424,E2 -21726.424} C_VEL
LIN {X 0,Y 216.348,Z 225.218,A -85,B 0,C 180,E1 -21727.453,E2 -21727.453} C_VEL
LIN {X 0,Y 210.227,Z 210.322,A -85,B 0,C 180,E1 -21729.369,E2 -21729.369} C_VEL
LIN {X 0,Y 203.789,Z 197.164,A -85,B 0,C 180,E1 -21731.456,E2 -21731.456} C_VEL
LIN {X 0,Y 199.028,Z 188.73,A -85,B 0,C 180,E1 -21733.071,E2 -21733.071} C_VEL
LIN {X 0,Y 196.515,Z 184.393,A -85,B 0,C 180,E1 -21733.967,E2 -21733.967} C_VEL
LIN {X 0,Y 194.092,Z 179.961,A -85,B 0,C 180,E1 -21734.899,E2 -21734.899} C_VEL
LIN {X 0,Y 192.504,Z 174.504,A -85,B 0,C 180,E1 -21738.613,E2 -21738.613} C_VEL
LIN {X 0,Y 192.577,Z 174.489,A -85,B 0,C 180,E1 -21743.403,E2 -21743.403} C_VEL
LIN {X 0,Y 192.6,Z 174.482,A -85,B 0,C 180,E1 -21747.06,E2 -21747.06} C_VEL
LIN {X 0,Y 192.613,Z 174.476,A -85,B 0,C 180,E1 -21751.684,E2 -21751.684} C_VEL
LIN {X 0,Y 192.656,Z 174.473,A -85,B 0,C 180,E1 -21756.342,E2 -21756.342} C_VEL
LIN {X 0,Y 192.688,Z 174.479,A -85,B 0,C 180,E1 -21761.491,E2 -21761.491} C_VEL
LIN {X 0,Y 192.767,Z 174.472,A -85,B 0,C 180,E1 -21767.364,E2 -21767.364} C_VEL
LIN {X 0,Y 193.011,Z 174.432,A -85,B 0,C 180,E1 -21771.625,E2 -21771.625} C_VEL
LIN {X 0,Y 193.218,Z 174.397,A -85,B 0,C 180,E1 -21777.916,E2 -21777.916} C_VEL
LIN {X 0,Y 193.405,Z 174.389,A -85,B 0,C 180,E1 -21780,E2 -21780} C_VEL
LIN {X 0,Y 192.927,Z 174.433,A -85,B 0,C 180,E1 -21784.178,E2 -21784.178} C_VEL
LIN {X 0,Y 193.019,Z 174.442,A -85,B 0,C 180,E1 -21788.375,E2 -21788.375} C_VEL
LIN {X 0,Y 192.748,Z 174.455,A -85,B 0,C 180,E1 -21792.637,E2 -21792.637} C_VEL
LIN {X 0,Y 192.698,Z 174.48,A -85,B 0,C 180,E1 -21796.964,E2 -21796.964} C_VEL
LIN {X 0,Y 192.574,Z 174.49,A -85,B 0,C 180,E1 -21801.405,E2 -21801.405} C_VEL
LIN {X 0,Y 192.625,Z 174.486,A -85,B 0,C 180,E1 -21804.203,E2 -21804.203} C_VEL
LIN {X 0,Y 192.596,Z 174.495,A -85,B 0,C 180,E1 -21808.866,E2 -21808.866} C_VEL
LIN {X 0,Y 192.59,Z 174.49,A -85,B 0,C 180,E1 -21813.188,E2 -21813.188} C_VEL
LIN {X 0,Y 192.537,Z 174.5,A -85,B 0,C 180,E1 -21818.356,E2 -21818.356} C_VEL
LIN {X 0,Y 192.482,Z 174.509,A -85,B 0,C 180,E1 -21823.095,E2 -21823.095} C_VEL
LIN {X 0,Y 192.563,Z 174.696,A -85,B 0,C 180,E1 -21824.956,E2 -21824.956} C_VEL
LIN {X 0,Y 193.585,Z 177.416,A -85,B 0,C 180,E1 -21825.401,E2 -21825.401} C_VEL
LIN {X 0,Y 195.713,Z 179.907,A -85,B 0,C 180,E1 -21826.143,E2 -21826.143} C_VEL
LIN {X 0,Y 197.879,Z 183.272,A -85,B 0,C 180,E1 -21826.913,E2 -21826.913} C_VEL
LIN {X 0,Y 204.085,Z 192.648,A -85,B 0,C 180,E1 -21828.969,E2 -21828.969} C_VEL
LIN {X 0,Y 211.14,Z 204.558,A -85,B 0,C 180,E1 -21831.144,E2 -21831.144} C_VEL
LIN {X 0,Y 215.325,Z 213.002,A -85,B 0,C 180,E1 -21832.395,E2 -21832.395} C_VEL
LIN {X 0,Y 219.283,Z 222.614,A -85,B 0,C 180,E1 -21833.581,E2 -21833.581} C_VEL
LIN {X 0,Y 216.717,Z 276.249,A -85,B 0,C 180,E1 -21835.276,E2 -21835.276} C_VEL
LIN {X 0,Y 215.439,Z 289.264,A -85,B 0,C 180,E1 -21836.002,E2 -21836.002} C_VEL
LIN {X 0,Y 213.514,Z 302.38,A -85,B 0,C 180,E1 -21837.106,E2 -21837.106} C_VEL
LIN {X 0,Y 211.419,Z 313.667,A -85,B 0,C 180,E1 -21838.43,E2 -21838.43} C_VEL
LIN {X 0,Y 208.595,Z 325.289,A -85,B 0,C 180,E1 -21840.203,E2 -21840.203} C_VEL
LIN {X 0,Y 205.736,Z 335.722,A -85,B 0,C 180,E1 -21842.263,E2 -21842.263} C_VEL
LIN {X 0,Y 203.062,Z 344.87,A -85,B 0,C 180,E1 -21844.564,E2 -21844.564} C_VEL
LIN {X 0,Y 200.063,Z 353.474,A -85,B 0,C 180,E1 -21847.27,E2 -21847.27} C_VEL
LIN {X 0,Y 197.305,Z 360.869,A -85,B 0,C 180,E1 -21850.223,E2 -21850.223} C_VEL
LIN {X 0,Y 195.058,Z 366.799,A -85,B 0,C 180,E1 -21853.249,E2 -21853.249} C_VEL
LIN {X 0,Y 193.273,Z 371.483,A -85,B 0,C 180,E1 -21856.33,E2 -21856.33} C_VEL
LIN {X 0,Y 191.923,Z 375.064,A -85,B 0,C 180,E1 -21859.451,E2 -21859.451} C_VEL
LIN {X 0,Y 191.354,Z 376.91,A -85,B 0,C 180,E1 -21861.553,E2 -21861.553} C_VEL
LIN {X 0,Y 190.86,Z 378.39,A -85,B 0,C 180,E1 -21863.836,E2 -21863.836} C_VEL
LIN {X 0,Y 190.466,Z 379.888,A -85,B 0,C 180,E1 -21867.887,E2 -21867.887} C_VEL
LIN {X 0,Y 190.417,Z 380.115,A -85,B 0,C 180,E1 -21870.001,E2 -21870.001} C_VEL
LIN {X 0,Y 190.465,Z 379.921,A -85,B 0,C 180,E1 -21872.116,E2 -21872.116} C_VEL
LIN {X 0,Y 190.89,Z 378.373,A -85,B 0,C 180,E1 -21876.342,E2 -21876.342} C_VEL
LIN {X 0,Y 191.354,Z 377.019,A -85,B 0,C 180,E1 -21878.449,E2 -21878.449} C_VEL
LIN {X 0,Y 192.295,Z 374.159,A -85,B 0,C 180,E1 -21881.597,E2 -21881.597} C_VEL
LIN {X 0,Y 193.777,Z 370.273,A -85,B 0,C 180,E1 -21884.708,E2 -21884.708} C_VEL
LIN {X 0,Y 195.734,Z 365.258,A -85,B 0,C 180,E1 -21887.771,E2 -21887.771} C_VEL
LIN {X 0,Y 198.086,Z 358.941,A -85,B 0,C 180,E1 -21890.782,E2 -21890.782} C_VEL
LIN {X 0,Y 201.035,Z 351.029,A -85,B 0,C 180,E1 -21893.706,E2 -21893.706} C_VEL
LIN {X 0,Y 203.867,Z 342.372,A -85,B 0,C 180,E1 -21896.26,E2 -21896.26} C_VEL
LIN {X 0,Y 206.903,Z 332.025,A -85,B 0,C 180,E1 -21898.672,E2 -21898.672} C_VEL
LIN {X 0,Y 209.907,Z 320.613,A -85,B 0,C 180,E1 -21900.704,E2 -21900.704} C_VEL
LIN {X 0,Y 212.425,Z 309.397,A -85,B 0,C 180,E1 -21902.242,E2 -21902.242} C_VEL
LIN {X 0,Y 214.437,Z 297.994,A -85,B 0,C 180,E1 -21903.437,E2 -21903.437} C_VEL
LIN {X 0,Y 216.081,Z 284.704,A -85,B 0,C 180,E1 -21904.428,E2 -21904.428} C_VEL
LIN {X 0,Y 217.183,Z 271.347,A -85,B 0,C 180,E1 -21905.033,E2 -21905.033} C_VEL
LIN {X 0,Y 219.483,Z 222.907,A -85,B 0,C 180,E1 -21906.529,E2 -21906.529} C_VEL
LIN {X 0,Y 213.957,Z 209.917,A -85,B 0,C 180,E1 -21908.186,E2 -21908.186} C_VEL
LIN {X 0,Y 208.7,Z 200.205,A -85,B 0,C 180,E1 -21909.766,E2 -21909.766} C_VEL
LIN {X 0,Y 201.004,Z 187.693,A -85,B 0,C 180,E1 -21912.223,E2 -21912.223} C_VEL
LIN {X 0,Y 195.813,Z 180.146,A -85,B 0,C 180,E1 -21914.006,E2 -21914.006} C_VEL
LIN {X 0,Y 194.899,Z 178.976,A -85,B 0,C 180,E1 -21914.328,E2 -21914.328} C_VEL
LIN {X 0,Y 193.139,Z 176.613,A -85,B 0,C 180,E1 -21914.966,E2 -21914.966} C_VEL
LIN {X 0,Y 192.522,Z 174.494,A -85,B 0,C 180,E1 -21915.344,E2 -21915.344} C_VEL
LIN {X 0,Y 192.506,Z 174.492,A -85,B 0,C 180,E1 -21920.056,E2 -21920.056} C_VEL
LIN {X 0,Y 192.559,Z 174.485,A -85,B 0,C 180,E1 -21924.27,E2 -21924.27} C_VEL
LIN {X 0,Y 192.606,Z 174.49,A -85,B 0,C 180,E1 -21927.061,E2 -21927.061} C_VEL
LIN {X 0,Y 192.622,Z 174.477,A -85,B 0,C 180,E1 -21931.685,E2 -21931.685} C_VEL
LIN {X 0,Y 192.677,Z 174.468,A -85,B 0,C 180,E1 -21936.345,E2 -21936.345} C_VEL
LIN {X 0,Y 192.696,Z 174.481,A -85,B 0,C 180,E1 -21941.491,E2 -21941.491} C_VEL
LIN {X 0,Y 192.778,Z 174.466,A -85,B 0,C 180,E1 -21947.365,E2 -21947.365} C_VEL
LIN {X 0,Y 193.024,Z 174.422,A -85,B 0,C 180,E1 -21951.626,E2 -21951.626} C_VEL
LIN {X 0,Y 193.229,Z 174.414,A -85,B 0,C 180,E1 -21957.916,E2 -21957.916} C_VEL
LIN {X 0,Y 193.413,Z 174.372,A -85,B 0,C 180,E1 -21960,E2 -21960} C_VEL
LIN {X 0,Y 192.927,Z 174.449,A -85,B 0,C 180,E1 -21964.178,E2 -21964.178} C_VEL
LIN {X 0,Y 193.018,Z 174.421,A -85,B 0,C 180,E1 -21968.375,E2 -21968.375} C_VEL
LIN {X 0,Y 192.752,Z 174.473,A -85,B 0,C 180,E1 -21972.637,E2 -21972.637} C_VEL
LIN {X 0,Y 192.681,Z 174.462,A -85,B 0,C 180,E1 -21976.966,E2 -21976.966} C_VEL
LIN {X 0,Y 192.572,Z 174.491,A -85,B 0,C 180,E1 -21981.405,E2 -21981.405} C_VEL
LIN {X 0,Y 192.611,Z 174.479,A -85,B 0,C 180,E1 -21984.188,E2 -21984.188} C_VEL
LIN {X 0,Y 192.601,Z 174.48,A -85,B 0,C 180,E1 -21988.865,E2 -21988.865} C_VEL
LIN {X 0,Y 192.595,Z 174.484,A -85,B 0,C 180,E1 -21993.186,E2 -21993.186} C_VEL
LIN {X 0,Y 192.542,Z 174.492,A -85,B 0,C 180,E1 -21998.354,E2 -21998.354} C_VEL
LIN {X 0,Y 192.544,Z 174.662,A -85,B 0,C 180,E1 -22001.534,E2 -22001.534} C_VEL
LIN {X 0,Y 194.215,Z 180.157,A -85,B 0,C 180,E1 -22005.065,E2 -22005.065} C_VEL
LIN {X 0,Y 196.527,Z 184.363,A -85,B 0,C 180,E1 -22005.937,E2 -22005.937} C_VEL
LIN {X 0,Y 198.221,Z 187.289,A -85,B 0,C 180,E1 -22006.548,E2 -22006.548} C_VEL
LIN {X 0,Y 203.366,Z 196.288,A -85,B 0,C 180,E1 -22008.312,E2 -22008.312} C_VEL
LIN {X 0,Y 208.962,Z 207.543,A -85,B 0,C 180,E1 -22010.147,E2 -22010.147} C_VEL
LIN {X 0,Y 215.177,Z 221.924,A -85,B 0,C 180,E1 -22012.1,E2 -22012.1} C_VEL
LIN {X 0,Y 216.674,Z 226.162,A -85,B 0,C 180,E1 -22012.578,E2 -22012.578} C_VEL
LIN {X 0,Y 218.235,Z 238.954,A -85,B 0,C 180,E1 -22013.402,E2 -22013.402} C_VEL
LIN {X 0,Y 218.23,Z 242.816,A -85,B 0,C 180,E1 -22013.556,E2 -22013.556} C_VEL
LIN {X 0,Y 217.65,Z 246.689,A -85,B 0,C 180,E1 -22013.599,E2 -22013.599} C_VEL
LIN {X 0,Y 215.478,Z 254.316,A -85,B 0,C 180,E1 -22013.485,E2 -22013.485} C_VEL
LIN {X 0,Y 212.475,Z 263.916,A -85,B 0,C 180,E1 -22013.285,E2 -22013.285} C_VEL
LIN {X 0,Y 211.518,Z 269.834,A -85,B 0,C 180,E1 -22013.338,E2 -22013.338} C_VEL
LIN {X 0,Y 210.315,Z 291.022,A -85,B 0,C 180,E1 -22014.07,E2 -22014.07} C_VEL
LIN {X 0,Y 208.718,Z 304.206,A -85,B 0,C 180,E1 -22014.84,E2 -22014.84} C_VEL
LIN {X 0,Y 206.616,Z 316.05,A -85,B 0,C 180,E1 -22015.857,E2 -22015.857} C_VEL
LIN {X 0,Y 204.104,Z 327.135,A -85,B 0,C 180,E1 -22017.157,E2 -22017.157} C_VEL
LIN {X 0,Y 201.079,Z 338.701,A -85,B 0,C 180,E1 -22018.966,E2 -22018.966} C_VEL
LIN {X 0,Y 197.843,Z 349.117,A -85,B 0,C 180,E1 -22021.052,E2 -22021.052} C_VEL
LIN {X 0,Y 194.97,Z 357.639,A -85,B 0,C 180,E1 -22023.218,E2 -22023.218} C_VEL
LIN {X 0,Y 192.233,Z 365.509,A -85,B 0,C 180,E1 -22025.713,E2 -22025.713} C_VEL
LIN {X 0,Y 189.482,Z 373.203,A -85,B 0,C 180,E1 -22028.799,E2 -22028.799} C_VEL
LIN {X 0,Y 187.485,Z 378.478,A -85,B 0,C 180,E1 -22031.419,E2 -22031.419} C_VEL
LIN {X 0,Y 185.46,Z 383.588,A -85,B 0,C 180,E1 -22034.616,E2 -22034.616} C_VEL
LIN {X 0,Y 184.228,Z 387.57,A -85,B 0,C 180,E1 -22037.887,E2 -22037.887} C_VEL
LIN {X 0,Y 183.426,Z 390.516,A -85,B 0,C 180,E1 -22041.183,E2 -22041.183} C_VEL
LIN {X 0,Y 183.075,Z 392.926,A -85,B 0,C 180,E1 -22045.596,E2 -22045.596} C_VEL
LIN {X 0,Y 183.122,Z 393.542,A -85,B 0,C 180,E1 -22047.799,E2 -22047.799} C_VEL
LIN {X 0,Y 183.268,Z 393.76,A -85,B 0,C 180,E1 -22049.999,E2 -22049.999} C_VEL
LIN {X 0,Y 183.087,Z 393.206,A -85,B 0,C 180,E1 -22053.584,E2 -22053.584} C_VEL
LIN {X 0,Y 183.184,Z 391.892,A -85,B 0,C 180,E1 -22056.608,E2 -22056.608} C_VEL
LIN {X 0,Y 183.441,Z 390.474,A -85,B 0,C 180,E1 -22058.814,E2 -22058.814} C_VEL
LIN {X 0,Y 184.23,Z 387.509,A -85,B 0,C 180,E1 -22062.11,E2 -22062.11} C_VEL
LIN {X 0,Y 185.458,Z 383.503,A -85,B 0,C 180,E1 -22065.381,E2 -22065.381} C_VEL
LIN {X 0,Y 187.809,Z 377.363,A -85,B 0,C 180,E1 -22069.112,E2 -22069.112} C_VEL
